// TIA Portal V19 program export: 0 tag tables, 0 data types, 3 data blocks, 24 code blocks (in call order from the OBs), 38 instance data blocks

DATA_BLOCK "time and date"   // DB89
{ S7_Optimized_Access := 'TRUE' }
// stored: MemoryReserve 100
   VAR RETAIN
      "Read time" : DTL;
      "write time" : DTL;
   END_VAR
   VAR
      "Set Time" : Bool;
      day : Int;
      month : Int;
      year : Int;
      hour : Int;
      minute : Int;
   END_VAR
   VAR RETAIN
      "Recipe Start Time" : DTL;
   END_VAR
BEGIN
END_DATA_BLOCK

DATA_BLOCK "IO Mapping"   // DB3
{ S7_Optimized_Access := 'TRUE' }
// stored: MemoryReserve 100
   VAR
      DI : Struct
         "Safety OK" : Bool;
         "IBC Valve is Open" : Bool;
         "IBC Valve is Closed" : Bool;
         "Pump Valve is Open" : Bool;
         "Pump Valve is Closed" : Bool;
         "Flowmeter Feed Valve is Open" : Bool;
         "Flowmerter Feed Valve is Closed" : Bool;
         "Dose Valve is Open" : Bool;
         "Dose Valve is Closed" : Bool;
         "DOL Running Feedback" : Bool;
         "Spare 11" : Bool;
         "Spare 12" : Bool;
         "Spare 13" : Bool;
         "Spare 14" : Bool;
      END_STRUCT;
      DQ : Struct
         "CMD Open IBC Valve" : Bool;
         "CMD Open Pump Feed Valve" : Bool;
         "CMD Open Flowmeter Feed Valve" : Bool;
         "CMD Opend Dosing Valve" : Bool;
         "Run Motor Cooling" : Bool;
         "Spare 6" : Bool;
         "Spare 7" : Bool;
         "Spare 8" : Bool;
         "Spare 9" : Bool;
         "Spare 10" : Bool;
      END_STRUCT;
      AI : Struct
         "Line Pressure" : Int;
         "Buffer level" : Int;
         "Spare 1" : Int;
         "Spare 2" : Int;
      END_STRUCT;
   END_VAR
BEGIN
END_DATA_BLOCK

DATA_BLOCK "HMI Tags"   // DB72
{ S7_Optimized_Access := 'TRUE' }
// stored: MemoryReserve 100
   VAR
      ControlAutoSelect : Bool := FALSE;
      ControlAutoStart : Bool := FALSE;
      ControlAutoStop : Bool := FALSE;
      AutoRunning : Bool := FALSE;
      ResetAlarms : Bool := FALSE;
   END_VAR
   VAR RETAIN
      "Select Input" : Struct
         "Input 1" : Int := 1;
         "Input 2" : Int := 10;
         "Input 3" : Int := 0;
         "Input 4" : Int := 0;
         "Input 5" : Int := 0;
         "Input 6" : Int := 0;
         "Input 7" : Int := 0;
         "Input 8" : Int := 0;
         "Input 9" : Int := 0;
         "Input 10" : Int := 0;
         "Input 11" : Int := 0;
         "Input 12" : Int := 0;
         "Input 13" : Int := 0;
         "Input 14" : Int := 0;
      END_STRUCT;
      "Selected Input" : Struct
         "Input 1" : Int := 0;
         "Input 2" : Int := 0;
         "Input 3" : Int := 0;
         "Input 4" : Int := 0;
         "Input 5" : Int := 0;
         "Input 6" : Int := 0;
         "Input 7" : Int := 0;
         "Input 8" : Int := 0;
         "Input 9" : Int := 0;
         "Input 10" : Int := 0;
         "Input 11" : Int := 0;
         "Input 12" : Int := 0;
         "Input 13" : Int := 0;
         "Input 14" : Int := 0;
      END_STRUCT;
      "Select Output" : Struct
         "output 1" : Int := 0;
         "output 2" : Int := 0;
         "output 3" : Int := 0;
         "output 4" : Int := 0;
         "output 5" : Int := 0;
         "output 6" : Int := 0;
         "output 7" : Int := 0;
         "output 8" : Int := 0;
         "output 9" : Int := 0;
         "output 10" : Int := 0;
      END_STRUCT;
      "Selected Output" : Struct
         "output 1" : Int := 0;
         "output 2" : Int := 0;
         "output 3" : Int := 0;
         "output 4" : Int := 0;
         "output 5" : Int := 0;
         "output 6" : Int := 0;
         "output 7" : Int := 0;
         "output 8" : Int := 0;
         "output 9" : Int := 0;
         "output 10" : Int := 0;
      END_STRUCT;
      LinePressure : "AnalogScale";
      BufferLevel { S7_SetPoint := 'True'} : "AnalogScale";
      SpareAN1 { S7_SetPoint := 'True'} : "AnalogScale";
      SpareAN2 { S7_SetPoint := 'True'} : "AnalogScale";
      CoolOverRunValue { S7_SetPoint := 'True'} : Time := T#1M;
      Pump_Control : "VFD_Control";
   END_VAR
   VAR
      ResetMotorFault : Bool := FALSE;
   END_VAR
   VAR RETAIN
      LinePressureMin { S7_SetPoint := 'True'} : Real := 0.0;
      LinePressureMax : Real := 0.0;
      LinePressureSP : Real := 0.0;
   END_VAR
   VAR
      "Manual Run Motor" : Bool := FALSE;
   END_VAR
   VAR RETAIN
      ModeOneShot : Bool := FALSE;
      ModeRepeat : Bool := TRUE;
      ModeOneShotTime : Bool := FALSE;
      ModeRepeatTime : Bool := FALSE;
      ModeContinous : Bool := FALSE;
   END_VAR
   VAR
      StartDose : Bool := FALSE;
   END_VAR
   VAR RETAIN
      "Required Dose" : Real := 1000.0;
      InflightVal : Real := 0.0;
      CalcDose : Real := 1000.0;
      DoseTime : Time := T#0MS;
      IntervalTime : Time := T#5S;
      IBC : "Valve";
      Flowmeter { S7_SetPoint := 'True'} : "Valve";
      Dose { S7_SetPoint := 'True'} : "Valve";
      Pump { S7_SetPoint := 'True'} : "Valve";
      WriteLogs { S7_SetPoint := 'True'} : Bool := FALSE;
   END_VAR
   VAR
      alarms : DWord := 16#0000_0000;
   END_VAR
   VAR RETAIN
      MinimumLinePressure : Real := 0.0;
      MaximumLinePressure : Real := 12.0;
      SystemEnables : Struct
         "Flowmeter Fitted" : Bool := TRUE;
         LinePressureFitted : Bool := TRUE;
         FlowmeterTemperatureFitted : Bool := TRUE;
         IBCFitted : Bool := FALSE;
         IBCValveFitted : Bool := FALSE;
         FlowmeterValveFitted : Bool := TRUE;
         "Buffer LevelFitted" : Bool := FALSE;
         PumpValveFitted : Bool := FALSE;
         DoseValveFitted : Bool := TRUE;
         ForcedCoolingFitted : Bool := TRUE;
         BufferValveFitted : Bool := FALSE;
      END_STRUCT;
      TemperatureLowSP : Real := 15.0;
      TemperatureHighSP : Real := 30.0;
      BufferHopperMinLVL : Real := 0.0;
      BufferHopperMaxLVL : Real := 0.0;
      BufferHopperLVLSP : Real := 0.0;
      HMISettingsLock : Bool := FALSE;
   END_VAR
   VAR
      DoseState : Int := 0;
   END_VAR
   VAR RETAIN
      DoseWaiting : Time := T#5S;
   END_VAR
   VAR
      FMActualCount : Real := 0.0;
      DoseActTime : Time := T#0MS;
      FmTemperature : Real := 17.8934;
   END_VAR
BEGIN
   LinePressure.AnalogMin := 0;
   LinePressure.AnalogMax := 27648;
   LinePressure.ScaledMIN := 0.0;
   LinePressure.ScaledMax := 11.0;
   LinePressure.ScaledSensor := 0.06127026;
   BufferLevel.AnalogMin := 0;
   BufferLevel.AnalogMax := 0;
   BufferLevel.ScaledMIN := 0.0;
   BufferLevel.ScaledMax := 0.0;
   BufferLevel.ScaledSensor := 0.0;
   SpareAN1.AnalogMin := 0;
   SpareAN1.AnalogMax := 0;
   SpareAN1.ScaledMIN := 0.0;
   SpareAN1.ScaledMax := 0.0;
   SpareAN1.ScaledSensor := 0.0;
   SpareAN2.AnalogMin := 0;
   SpareAN2.AnalogMax := 0;
   SpareAN2.ScaledMIN := 0.0;
   SpareAN2.ScaledMax := 0.0;
   SpareAN2.ScaledSensor := 0.0;
   Pump_Control.NameplateSpeed := 710.0;
   Pump_Control.AutoSpeedSP := 50.0;
   Pump_Control.DriveIsRunning := FALSE;
   Pump_Control.ActualSpeed := 0.0;
   Pump_Control.AxisActive := FALSE;
   Pump_Control.LockoutActive := FALSE;
   Pump_Control.ErrorPResent := FALSE;
   Pump_Control.HMI_VFD_Fault := 0;
   Pump_Control.HMI_Error_Present := FALSE;
   Pump_Control.VFDFaultCode := 0;
   Pump_Control.MotorState := 0;
   Pump_Control.Actual_Current := 0.0007141113;
   Pump_Control.Actual_torque := 0.0;
   Pump_Control.Peak_Current := 0.0;
   Pump_Control.Peak_torque := 0.0;
   IBC.ManOpen := FALSE;
   IBC.FeebackFitted := FALSE;
   IBC.ValveisOpen := FALSE;
   IBC.ValveisClosed := FALSE;
   IBC.ValveAngle := 0.0;
   IBC.FeedbackFaultTime := T#0MS;
   Flowmeter.ManOpen := FALSE;
   Flowmeter.FeebackFitted := FALSE;
   Flowmeter.ValveisOpen := FALSE;
   Flowmeter.ValveisClosed := TRUE;
   Flowmeter.ValveAngle := 90.0;
   Flowmeter.FeedbackFaultTime := T#0MS;
   Dose.ManOpen := FALSE;
   Dose.FeebackFitted := FALSE;
   Dose.ValveisOpen := FALSE;
   Dose.ValveisClosed := TRUE;
   Dose.ValveAngle := 90.0;
   Dose.FeedbackFaultTime := T#0MS;
   Pump.ManOpen := FALSE;
   Pump.FeebackFitted := FALSE;
   Pump.ValveisOpen := FALSE;
   Pump.ValveisClosed := FALSE;
   Pump.ValveAngle := 0.0;
   Pump.FeedbackFaultTime := T#0MS;
END_DATA_BLOCK

ORGANIZATION_BLOCK "Main"   // OB1, LAD, ProgramCycle
TITLE = "Main Program Sweep (Cycle)"
{ S7_Optimized_Access := 'TRUE' }
// stored: SetENOAutomatically false
   VAR_INPUT
      Initial_Call : Bool;   // Initial call of this OB
      Remanence : Bool;   // =True, if remanent data are available
   END_VAR
   VAR_TEMP   // added for the SCL form of the ladder/FBD networks
      _w1 : Bool;
   END_VAR
BEGIN

REGION Network 1: Control
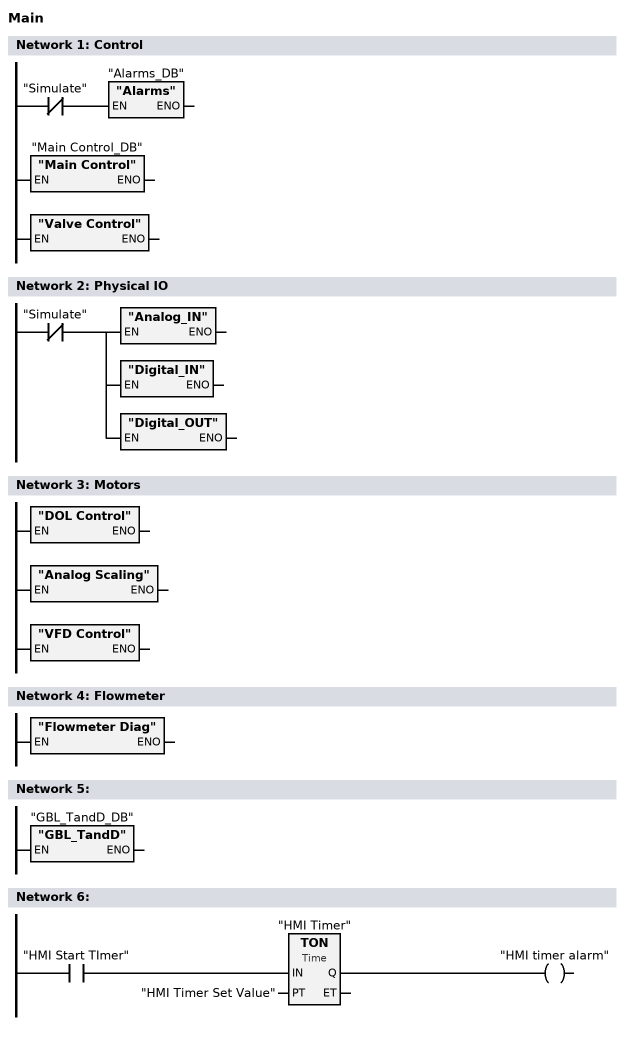
   RUNG wire#powerrail
      I_Contact( "Simulate" )
      "Alarms_DB"()
   END_RUNG
   RUNG wire#powerrail
      "Main Control_DB"()
   END_RUNG
   RUNG wire#powerrail
      "Valve Control"()
   END_RUNG
   // the same network as SCL:
   IF NOT "Simulate" THEN
       "Alarms_DB"();   // "Alarms"
   END_IF;
   "Main Control_DB"();   // "Main Control"
   "Valve Control"();
END_REGION

REGION Network 2: Physical IO
   RUNG wire#powerrail
      I_Contact( "Simulate" )
      wire#w1
      "Analog_IN"()
   END_RUNG
   RUNG wire#w1
      "Digital_IN"()
   END_RUNG
   RUNG wire#w1
      "Digital_OUT"()
   END_RUNG
   // the same network as SCL:
   #_w1 := NOT "Simulate";
   IF #_w1 THEN
       "Analog_IN"();
       "Digital_IN"();
       "Digital_OUT"();
   END_IF;
END_REGION

REGION Network 3: Motors
   RUNG wire#powerrail
      "DOL Control"()
   END_RUNG
   RUNG wire#powerrail
      "Analog Scaling"()
   END_RUNG
   RUNG wire#powerrail
      "VFD Control"()
   END_RUNG
   // the same network as SCL:
   "DOL Control"();
   "Analog Scaling"();
   "VFD Control"();
END_REGION

REGION Network 4: Flowmeter
   RUNG wire#powerrail
      "Flowmeter Diag"()
   END_RUNG
   // the same network as SCL:
   "Flowmeter Diag"();
END_REGION

REGION Network 5
   RUNG wire#powerrail
      "GBL_TandD_DB"()
   END_RUNG
   // the same network as SCL:
   "GBL_TandD_DB"();   // "GBL_TandD"
END_REGION

REGION Network 6
   RUNG wire#powerrail
      Contact( "HMI Start TImer" )
      { S7_Templates := "time_type := Time" } "HMI Timer".TON(pt := "HMI Timer Set Value", et =>)
      Coil( "HMI timer alarm" )
   END_RUNG
   // the same network as SCL:
   "HMI Timer".TON(IN := "HMI Start TImer", PT := "HMI Timer Set Value");
   "HMI timer alarm" := "HMI Timer".Q;
END_REGION
END_ORGANIZATION_BLOCK

FUNCTION_BLOCK "Alarms"   // FB7, LAD
{ S7_Optimized_Access := 'TRUE' }
// stored: MemoryReserve 100, SetENOAutomatically false
   VAR_TEMP   // added for the SCL form of the ladder/FBD networks
      _w1 : Bool;
      _w2 : Bool;
      _w3 : Bool;
   END_VAR
BEGIN

REGION Network 1: IBC Valve Open Fault
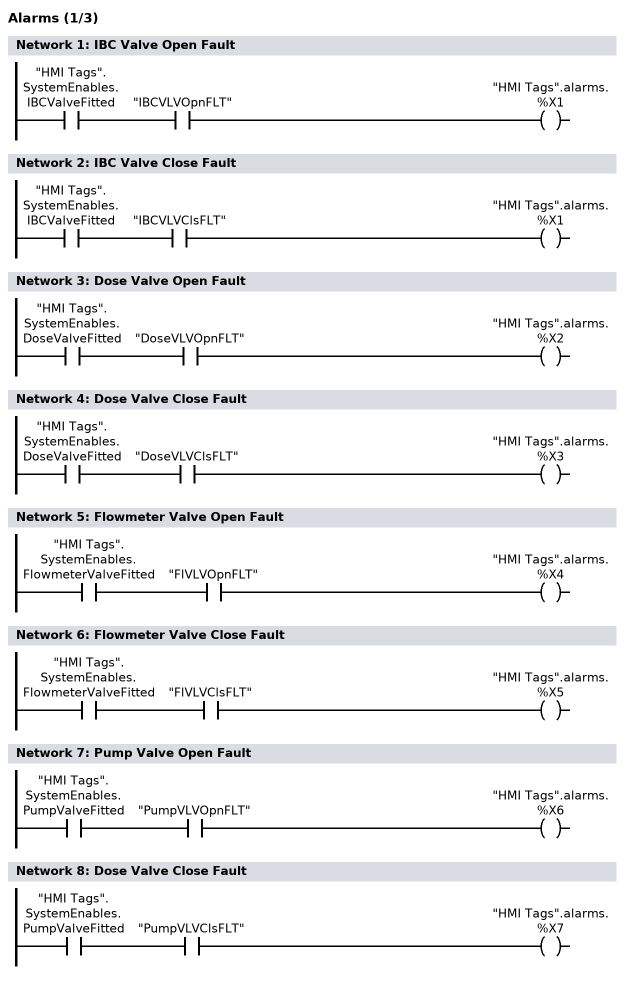
   RUNG wire#powerrail
      Contact( "HMI Tags".SystemEnables.IBCValveFitted )
      Contact( "IBCVLVOpnFLT" )
      Coil( "HMI Tags".alarms.%X1 )
   END_RUNG
   // the same network as SCL:
   "HMI Tags".alarms.%X1 := "HMI Tags".SystemEnables.IBCValveFitted AND "IBCVLVOpnFLT";
END_REGION

REGION Network 2: IBC Valve Close Fault
   RUNG wire#powerrail
      Contact( "HMI Tags".SystemEnables.IBCValveFitted )
      Contact( "IBCVLVClsFLT" )
      Coil( "HMI Tags".alarms.%X1 )
   END_RUNG
   // the same network as SCL:
   "HMI Tags".alarms.%X1 := "HMI Tags".SystemEnables.IBCValveFitted AND "IBCVLVClsFLT";
END_REGION

REGION Network 3: Dose Valve Open Fault
   RUNG wire#powerrail
      Contact( "HMI Tags".SystemEnables.DoseValveFitted )
      Contact( "DoseVLVOpnFLT" )
      Coil( "HMI Tags".alarms.%X2 )
   END_RUNG
   // the same network as SCL:
   "HMI Tags".alarms.%X2 := "HMI Tags".SystemEnables.DoseValveFitted AND "DoseVLVOpnFLT";
END_REGION

REGION Network 4: Dose Valve Close Fault
   RUNG wire#powerrail
      Contact( "HMI Tags".SystemEnables.DoseValveFitted )
      Contact( "DoseVLVClsFLT" )
      Coil( "HMI Tags".alarms.%X3 )
   END_RUNG
   // the same network as SCL:
   "HMI Tags".alarms.%X3 := "HMI Tags".SystemEnables.DoseValveFitted AND "DoseVLVClsFLT";
END_REGION

REGION Network 5: Flowmeter Valve Open Fault
   RUNG wire#powerrail
      Contact( "HMI Tags".SystemEnables.FlowmeterValveFitted )
      Contact( "FlVLVOpnFLT" )
      Coil( "HMI Tags".alarms.%X4 )
   END_RUNG
   // the same network as SCL:
   "HMI Tags".alarms.%X4 := "HMI Tags".SystemEnables.FlowmeterValveFitted AND "FlVLVOpnFLT";
END_REGION

REGION Network 6: Flowmeter Valve Close Fault
   RUNG wire#powerrail
      Contact( "HMI Tags".SystemEnables.FlowmeterValveFitted )
      Contact( "FlVLVClsFLT" )
      Coil( "HMI Tags".alarms.%X5 )
   END_RUNG
   // the same network as SCL:
   "HMI Tags".alarms.%X5 := "HMI Tags".SystemEnables.FlowmeterValveFitted AND "FlVLVClsFLT";
END_REGION

REGION Network 7: Pump Valve Open Fault
   RUNG wire#powerrail
      Contact( "HMI Tags".SystemEnables.PumpValveFitted )
      Contact( "PumpVLVOpnFLT" )
      Coil( "HMI Tags".alarms.%X6 )
   END_RUNG
   // the same network as SCL:
   "HMI Tags".alarms.%X6 := "HMI Tags".SystemEnables.PumpValveFitted AND "PumpVLVOpnFLT";
END_REGION

REGION Network 8: Dose Valve Close Fault
   RUNG wire#powerrail
      Contact( "HMI Tags".SystemEnables.PumpValveFitted )
      Contact( "PumpVLVClsFLT" )
      Coil( "HMI Tags".alarms.%X7 )
   END_RUNG
   // the same network as SCL:
   "HMI Tags".alarms.%X7 := "HMI Tags".SystemEnables.PumpValveFitted AND "PumpVLVClsFLT";
END_REGION

REGION Network 9: Flowmeter not counting when required
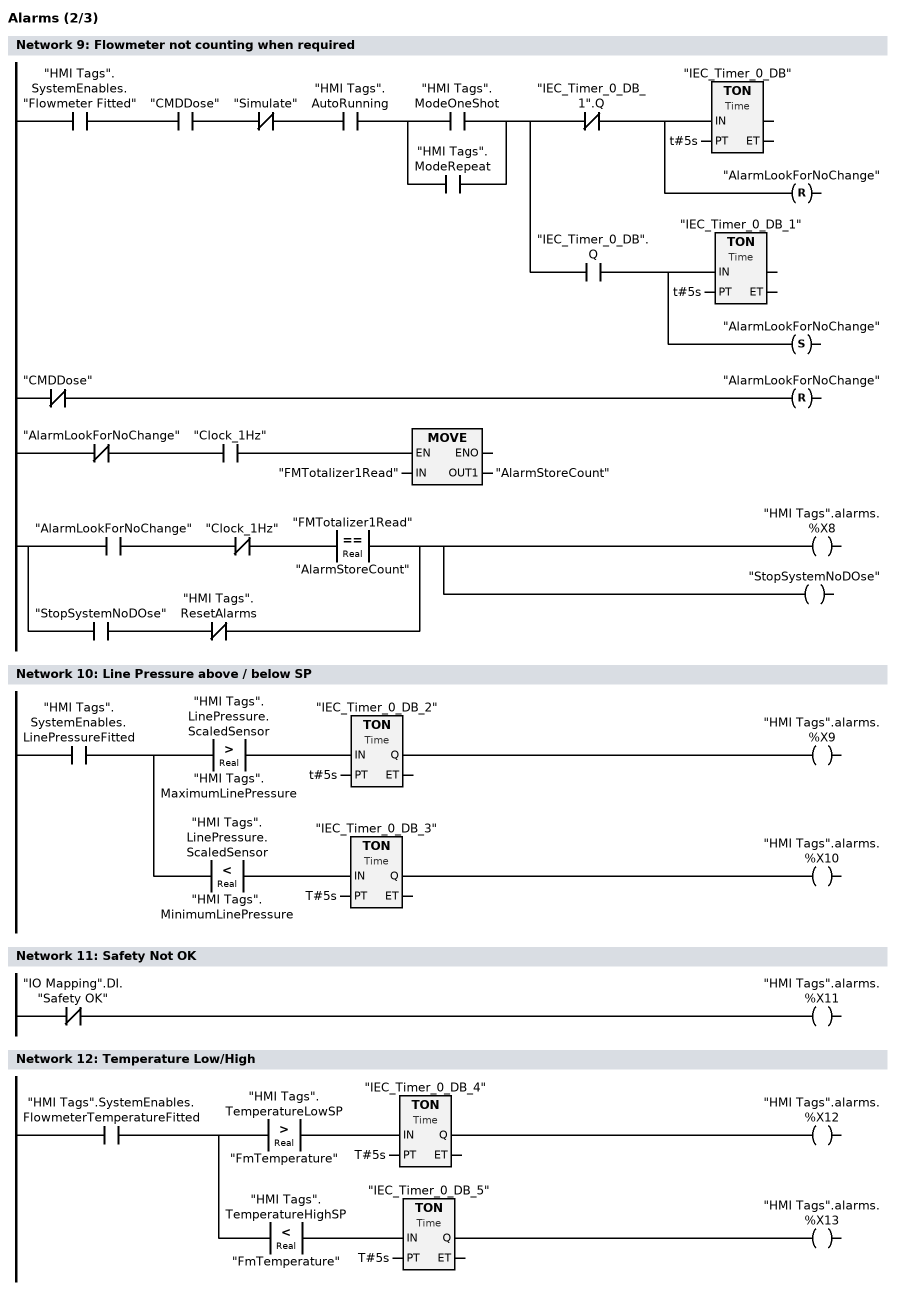
   RUNG wire#powerrail
      Contact( "HMI Tags".SystemEnables."Flowmeter Fitted" )
      Contact( "CMDDose" )
      I_Contact( "Simulate" )
      Contact( "HMI Tags".AutoRunning )
      wire#w1
      Contact( "HMI Tags".ModeOneShot )
      wire#w2
      I_Contact( "IEC_Timer_0_DB_1".Q )
      wire#w3
      { S7_Templates := "time_type := Time" } "IEC_Timer_0_DB".TON(pt := t#5s, et =>)
   END_RUNG
   RUNG wire#w1
      Contact( "HMI Tags".ModeRepeat )
   END_RUNG wire#w2
   RUNG wire#w3
      R_Coil( "AlarmLookForNoChange" )
   END_RUNG
   RUNG wire#w2
      Contact( "IEC_Timer_0_DB".Q )
      wire#w4
      { S7_Templates := "time_type := Time" } "IEC_Timer_0_DB_1".TON(pt := t#5s, et =>)
   END_RUNG
   RUNG wire#w4
      S_Coil( "AlarmLookForNoChange" )
   END_RUNG
   RUNG wire#powerrail
      I_Contact( "CMDDose" )
      R_Coil( "AlarmLookForNoChange" )
   END_RUNG
   RUNG wire#powerrail
      I_Contact( "AlarmLookForNoChange" )
      Contact( "Clock_1Hz" )
      Move(in := "FMTotalizer1Read", out1 => "AlarmStoreCount")
   END_RUNG
   RUNG wire#powerrail
      Contact( "AlarmLookForNoChange" )
      I_Contact( "Clock_1Hz" )
      { S7_Templates := "SrcType := Real" } EQ_Contact(in1 := "FMTotalizer1Read", in2 := "AlarmStoreCount")
      wire#w5
      Coil( "HMI Tags".alarms.%X8 )
   END_RUNG
   RUNG wire#powerrail
      Contact( "StopSystemNoDOse" )
      I_Contact( "HMI Tags".ResetAlarms )
   END_RUNG wire#w5
   RUNG wire#w5
      Coil( "StopSystemNoDOse" )
   END_RUNG
   // the same network as SCL:
   #_w1 := "HMI Tags".SystemEnables."Flowmeter Fitted" AND "CMDDose" AND NOT "Simulate" AND "HMI Tags".AutoRunning AND ("HMI Tags".ModeOneShot OR "HMI Tags".ModeRepeat);
   #_w2 := #_w1 AND NOT "IEC_Timer_0_DB_1".Q;
   "IEC_Timer_0_DB".TON(IN := #_w2, PT := t#5s);
   IF #_w2 THEN "AlarmLookForNoChange" := FALSE; END_IF;
   #_w3 := #_w1 AND "IEC_Timer_0_DB".Q;
   "IEC_Timer_0_DB_1".TON(IN := #_w3, PT := t#5s);
   IF #_w3 THEN "AlarmLookForNoChange" := TRUE; END_IF;
   IF NOT "CMDDose" THEN "AlarmLookForNoChange" := FALSE; END_IF;
   IF NOT "AlarmLookForNoChange" AND "Clock_1Hz" THEN "AlarmStoreCount" := "FMTotalizer1Read"; END_IF;
   "HMI Tags".alarms.%X8 := ("AlarmLookForNoChange" AND NOT "Clock_1Hz" AND ("FMTotalizer1Read" = "AlarmStoreCount")) OR ("StopSystemNoDOse" AND NOT "HMI Tags".ResetAlarms);
   "StopSystemNoDOse" := "HMI Tags".alarms.%X8;
END_REGION

REGION Network 10: Line Pressure above / below SP
   RUNG wire#powerrail
      Contact( "HMI Tags".SystemEnables.LinePressureFitted )
      wire#w1
      { S7_Templates := "SrcType := Real" } GT_Contact(in1 := "HMI Tags".LinePressure.ScaledSensor, in2 := "HMI Tags".MaximumLinePressure)
      { S7_Templates := "time_type := Time" } "IEC_Timer_0_DB_2".TON(pt := t#5s, et =>)
      Coil( "HMI Tags".alarms.%X9 )
   END_RUNG
   RUNG wire#w1
      { S7_Templates := "SrcType := Real" } LT_Contact(in1 := "HMI Tags".LinePressure.ScaledSensor, in2 := "HMI Tags".MinimumLinePressure)
      { S7_Templates := "time_type := Time" } "IEC_Timer_0_DB_3".TON(pt := T#5s, et =>)
      Coil( "HMI Tags".alarms.%X10 )
   END_RUNG
   // the same network as SCL:
   "IEC_Timer_0_DB_2".TON(IN := "HMI Tags".SystemEnables.LinePressureFitted AND ("HMI Tags".LinePressure.ScaledSensor > "HMI Tags".MaximumLinePressure),
                          PT := t#5s);
   "HMI Tags".alarms.%X9 := "IEC_Timer_0_DB_2".Q;
   "IEC_Timer_0_DB_3".TON(IN := "HMI Tags".SystemEnables.LinePressureFitted AND ("HMI Tags".LinePressure.ScaledSensor < "HMI Tags".MinimumLinePressure),
                          PT := T#5s);
   "HMI Tags".alarms.%X10 := "IEC_Timer_0_DB_3".Q;
END_REGION

REGION Network 11: Safety Not OK
   RUNG wire#powerrail
      I_Contact( "IO Mapping".DI."Safety OK" )
      Coil( "HMI Tags".alarms.%X11 )
   END_RUNG
   // the same network as SCL:
   "HMI Tags".alarms.%X11 := NOT "IO Mapping".DI."Safety OK";
END_REGION

REGION Network 12: Temperature Low/High
   RUNG wire#powerrail
      Contact( "HMI Tags".SystemEnables.FlowmeterTemperatureFitted )
      wire#w1
      { S7_Templates := "SrcType := Real" } GT_Contact(in1 := "HMI Tags".TemperatureLowSP, in2 := "FmTemperature")
      { S7_Templates := "time_type := Time" } "IEC_Timer_0_DB_4".TON(pt := T#5s, et =>)
      Coil( "HMI Tags".alarms.%X12 )
   END_RUNG
   RUNG wire#w1
      { S7_Templates := "SrcType := Real" } LT_Contact(in1 := "HMI Tags".TemperatureHighSP, in2 := "FmTemperature")
      { S7_Templates := "time_type := Time" } "IEC_Timer_0_DB_5".TON(pt := T#5s, et =>)
      Coil( "HMI Tags".alarms.%X13 )
   END_RUNG
   // the same network as SCL:
   "IEC_Timer_0_DB_4".TON(IN := "HMI Tags".SystemEnables.FlowmeterTemperatureFitted AND ("HMI Tags".TemperatureLowSP > "FmTemperature"),
                          PT := T#5s);
   "HMI Tags".alarms.%X12 := "IEC_Timer_0_DB_4".Q;
   "IEC_Timer_0_DB_5".TON(IN := "HMI Tags".SystemEnables.FlowmeterTemperatureFitted AND ("HMI Tags".TemperatureHighSP < "FmTemperature"),
                          PT := T#5s);
   "HMI Tags".alarms.%X13 := "IEC_Timer_0_DB_5".Q;
END_REGION

REGION Network 13: VFDFAULT
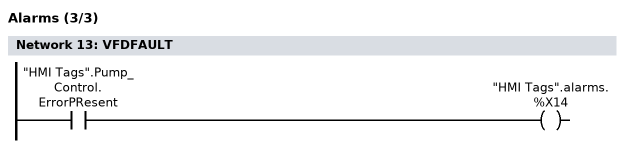
   RUNG wire#powerrail
      Contact( "HMI Tags".Pump_Control.ErrorPResent )
      Coil( "HMI Tags".alarms.%X14 )
   END_RUNG
   // the same network as SCL:
   "HMI Tags".alarms.%X14 := "HMI Tags".Pump_Control.ErrorPResent;
END_REGION
END_FUNCTION_BLOCK

FUNCTION_BLOCK "Main Control"   // FB1, LAD
{ S7_Optimized_Access := 'TRUE' }
// stored: MemoryReserve 100, SetENOAutomatically false
   VAR
      store : Bool;
   END_VAR
   VAR_TEMP   // added for the SCL form of the ladder/FBD networks
      _w1 : Bool;
      _w2 : Bool;
   END_VAR
BEGIN

REGION Network 1: Control Auto Run
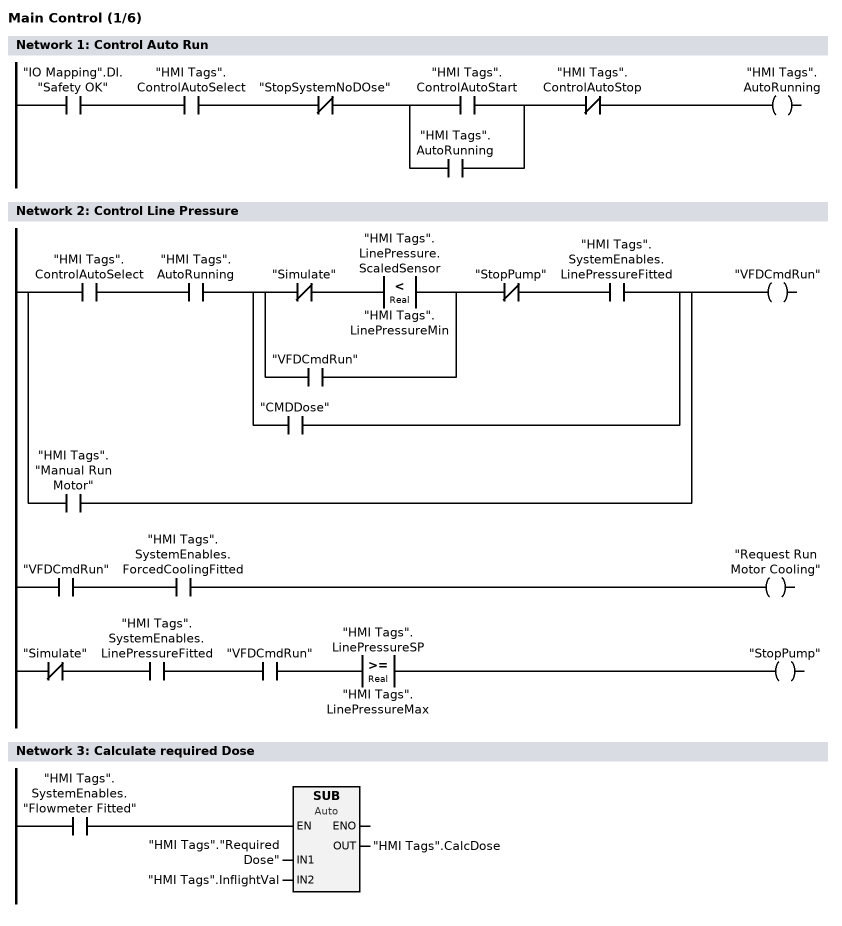
   RUNG wire#powerrail
      Contact( "IO Mapping".DI."Safety OK" )
      Contact( "HMI Tags".ControlAutoSelect )
      I_Contact( "StopSystemNoDOse" )
      wire#w1
      Contact( "HMI Tags".ControlAutoStart )
      wire#w2
      I_Contact( "HMI Tags".ControlAutoStop )
      Coil( "HMI Tags".AutoRunning )
   END_RUNG
   RUNG wire#w1
      Contact( "HMI Tags".AutoRunning )
   END_RUNG wire#w2
   // the same network as SCL:
   "HMI Tags".AutoRunning := "IO Mapping".DI."Safety OK" AND "HMI Tags".ControlAutoSelect AND NOT "StopSystemNoDOse" AND ("HMI Tags".ControlAutoStart OR "HMI Tags".AutoRunning) AND NOT "HMI Tags".ControlAutoStop;
END_REGION

REGION Network 2: Control Line Pressure
   RUNG wire#powerrail
      Contact( "HMI Tags".ControlAutoSelect )
      Contact( "HMI Tags".AutoRunning )
      wire#w1
      I_Contact( "Simulate" )
      { S7_Templates := "SrcType := Real" } LT_Contact(in1 := "HMI Tags".LinePressure.ScaledSensor, in2 := "HMI Tags".LinePressureMin)
      wire#w2
      I_Contact( "StopPump" )
      Contact( "HMI Tags".SystemEnables.LinePressureFitted )
      wire#w3
      Coil( "VFDCmdRun" )
   END_RUNG
   RUNG wire#w1
      Contact( "VFDCmdRun" )
   END_RUNG wire#w2
   RUNG wire#w1
      Contact( "CMDDose" )
   END_RUNG wire#w3
   RUNG wire#powerrail
      Contact( "HMI Tags"."Manual Run Motor" )
   END_RUNG wire#w3
   RUNG wire#powerrail
      Contact( "VFDCmdRun" )
      Contact( "HMI Tags".SystemEnables.ForcedCoolingFitted )
      Coil( "Request Run Motor Cooling" )
   END_RUNG
   RUNG wire#powerrail
      I_Contact( "Simulate" )
      Contact( "HMI Tags".SystemEnables.LinePressureFitted )
      Contact( "VFDCmdRun" )
      { S7_Templates := "SrcType := Real" } GE_Contact(in1 := "HMI Tags".LinePressureSP, in2 := "HMI Tags".LinePressureMax)
      Coil( "StopPump" )
   END_RUNG
   // the same network as SCL:
   "VFDCmdRun" := ("HMI Tags".ControlAutoSelect AND "HMI Tags".AutoRunning AND ((((NOT "Simulate" AND ("HMI Tags".LinePressure.ScaledSensor < "HMI Tags".LinePressureMin)) OR "VFDCmdRun") AND NOT "StopPump" AND "HMI Tags".SystemEnables.LinePressureFitted) OR "CMDDose")) OR "HMI Tags"."Manual Run Motor";
   "Request Run Motor Cooling" := "VFDCmdRun" AND "HMI Tags".SystemEnables.ForcedCoolingFitted;
   "StopPump" := NOT "Simulate" AND "HMI Tags".SystemEnables.LinePressureFitted AND "VFDCmdRun" AND ("HMI Tags".LinePressureSP >= "HMI Tags".LinePressureMax);
END_REGION

REGION Network 3: Calculate required Dose
   RUNG wire#powerrail
      Contact( "HMI Tags".SystemEnables."Flowmeter Fitted" )
      Sub(in1 := "HMI Tags"."Required Dose", in2 := "HMI Tags".InflightVal, out => "HMI Tags".CalcDose)
   END_RUNG
   // the same network as SCL:
   IF "HMI Tags".SystemEnables."Flowmeter Fitted" THEN
       "HMI Tags".CalcDose := "HMI Tags"."Required Dose" - "HMI Tags".InflightVal;
   END_IF;
END_REGION

REGION Network 4: Open Valves to Dose
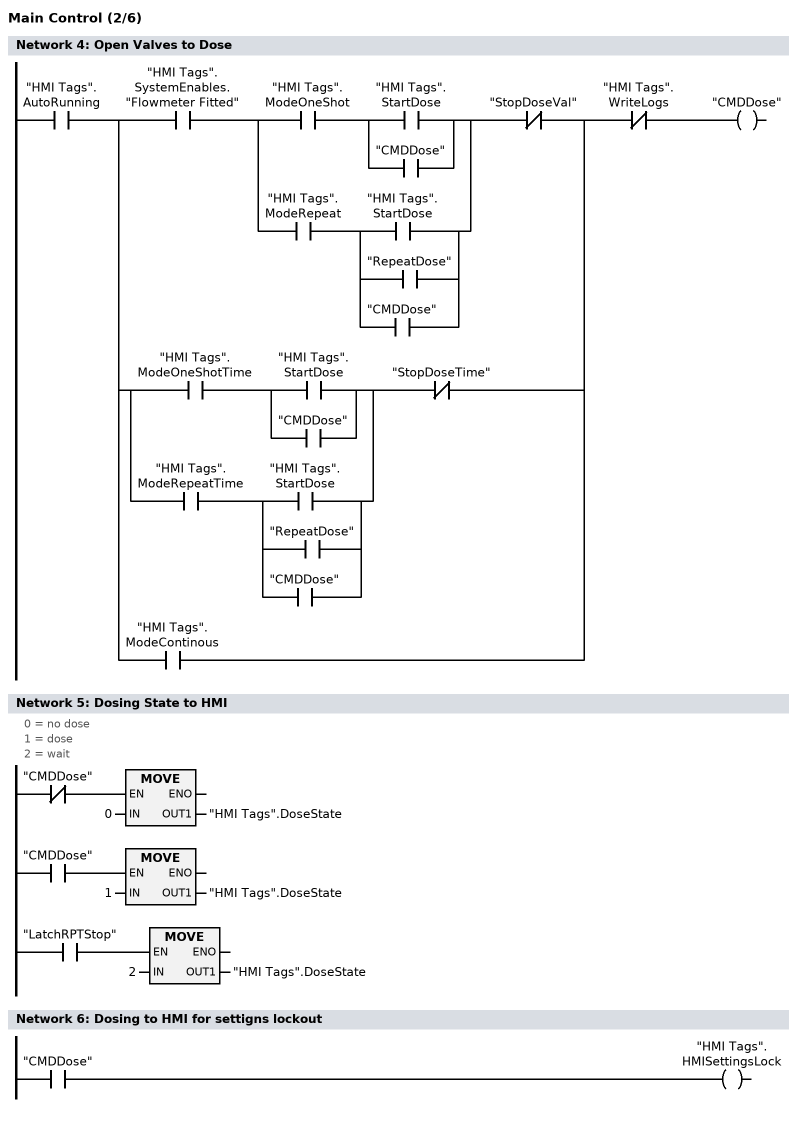
   RUNG wire#powerrail
      Contact( "HMI Tags".AutoRunning )
      wire#w1
      Contact( "HMI Tags".SystemEnables."Flowmeter Fitted" )
      wire#w2
      Contact( "HMI Tags".ModeOneShot )
      wire#w3
      Contact( "HMI Tags".StartDose )
      wire#w4
      I_Contact( "StopDoseVal" )
      wire#w6
      I_Contact( "HMI Tags".WriteLogs )
      Coil( "CMDDose" )
   END_RUNG
   RUNG wire#w3
      Contact( "CMDDose" )
   END_RUNG wire#w4
   RUNG wire#w2
      Contact( "HMI Tags".ModeRepeat )
      wire#w5
      Contact( "HMI Tags".StartDose )
   END_RUNG wire#w4
   RUNG wire#w5
      Contact( "RepeatDose" )
   END_RUNG wire#w4
   RUNG wire#w5
      Contact( "CMDDose" )
   END_RUNG wire#w4
   RUNG wire#w1
      Contact( "HMI Tags".ModeOneShotTime )
      wire#w7
      Contact( "HMI Tags".StartDose )
      wire#w8
      I_Contact( "StopDoseTime" )
   END_RUNG wire#w6
   RUNG wire#w7
      Contact( "CMDDose" )
   END_RUNG wire#w8
   RUNG wire#w1
      Contact( "HMI Tags".ModeRepeatTime )
      wire#w9
      Contact( "HMI Tags".StartDose )
   END_RUNG wire#w8
   RUNG wire#w9
      Contact( "RepeatDose" )
   END_RUNG wire#w8
   RUNG wire#w9
      Contact( "CMDDose" )
   END_RUNG wire#w8
   RUNG wire#w1
      Contact( "HMI Tags".ModeContinous )
   END_RUNG wire#w6
   // the same network as SCL:
   "CMDDose" := "HMI Tags".AutoRunning AND (("HMI Tags".SystemEnables."Flowmeter Fitted" AND (("HMI Tags".ModeOneShot AND ("HMI Tags".StartDose OR "CMDDose")) OR ("HMI Tags".ModeRepeat AND ("HMI Tags".StartDose OR "RepeatDose" OR "CMDDose"))) AND NOT "StopDoseVal") OR ((("HMI Tags".ModeOneShotTime AND ("HMI Tags".StartDose OR "CMDDose")) OR ("HMI Tags".ModeRepeatTime AND ("HMI Tags".StartDose OR "RepeatDose" OR "CMDDose"))) AND NOT "StopDoseTime") OR "HMI Tags".ModeContinous) AND NOT "HMI Tags".WriteLogs;
END_REGION

REGION Network 5: Dosing State to HMI
   // 0 = no dose
   // 1 = dose
   // 2 = wait
   RUNG wire#powerrail
      I_Contact( "CMDDose" )
      Move(in := 0, out1 => "HMI Tags".DoseState)
   END_RUNG
   RUNG wire#powerrail
      Contact( "CMDDose" )
      Move(in := 1, out1 => "HMI Tags".DoseState)
   END_RUNG
   RUNG wire#powerrail
      Contact( "LatchRPTStop" )
      Move(in := 2, out1 => "HMI Tags".DoseState)
   END_RUNG
   // the same network as SCL:
   IF NOT "CMDDose" THEN "HMI Tags".DoseState := 0; END_IF;
   IF "CMDDose" THEN "HMI Tags".DoseState := 1; END_IF;
   IF "LatchRPTStop" THEN "HMI Tags".DoseState := 2; END_IF;
END_REGION

REGION Network 6: Dosing to HMI for settigns lockout
   RUNG wire#powerrail
      Contact( "CMDDose" )
      Coil( "HMI Tags".HMISettingsLock )
   END_RUNG
   // the same network as SCL:
   "HMI Tags".HMISettingsLock := "CMDDose";
END_REGION

REGION Network 7: Command the flowmeter to count
   // This should start the flowmeter counting slightly ahead of opening the valves.
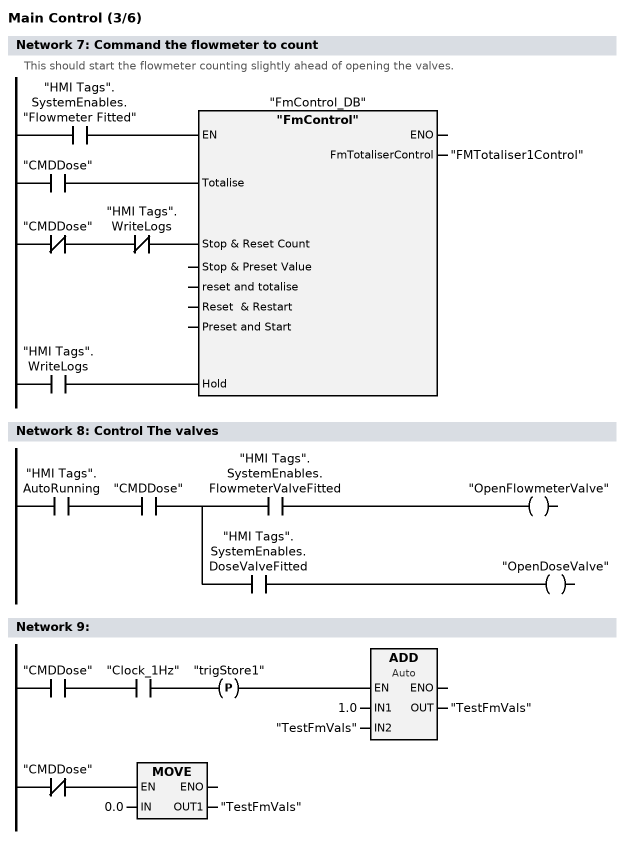
   RUNG wire#powerrail
      Contact( "HMI Tags".SystemEnables."Flowmeter Fitted" )
      "FmControl_DB"(Totalise := wire#w1, "Stop & Reset Count" := wire#w2, Hold := wire#w3, "Stop & Preset Value" :=, "reset and totalise" :=, "Reset  & Restart" :=, "Preset and Start" :=, FmTotaliserControl => "FMTotaliser1Control")
   END_RUNG
   RUNG wire#powerrail
      Contact( "CMDDose" )
   END_RUNG wire#w1
   RUNG wire#powerrail
      I_Contact( "CMDDose" )
      I_Contact( "HMI Tags".WriteLogs )
   END_RUNG wire#w2
   RUNG wire#powerrail
      Contact( "HMI Tags".WriteLogs )
   END_RUNG wire#w3
   // the same network as SCL:
   IF "HMI Tags".SystemEnables."Flowmeter Fitted" THEN
       "FmControl_DB"(Totalise := "CMDDose",   // "FmControl"
                      "Stop & Reset Count" := NOT "CMDDose" AND NOT "HMI Tags".WriteLogs,
                      Hold := "HMI Tags".WriteLogs,
                      FmTotaliserControl => "FMTotaliser1Control");
   END_IF;
END_REGION

REGION Network 8: Control The valves
   RUNG wire#powerrail
      Contact( "HMI Tags".AutoRunning )
      Contact( "CMDDose" )
      wire#w1
      Contact( "HMI Tags".SystemEnables.FlowmeterValveFitted )
      Coil( "OpenFlowmeterValve" )
   END_RUNG
   RUNG wire#w1
      Contact( "HMI Tags".SystemEnables.DoseValveFitted )
      Coil( "OpenDoseValve" )
   END_RUNG
   // the same network as SCL:
   #_w1 := "HMI Tags".AutoRunning AND "CMDDose";
   "OpenFlowmeterValve" := #_w1 AND "HMI Tags".SystemEnables.FlowmeterValveFitted;
   "OpenDoseValve" := #_w1 AND "HMI Tags".SystemEnables.DoseValveFitted;
END_REGION

REGION Network 9
   RUNG wire#powerrail
      Contact( "CMDDose" )
      Contact( "Clock_1Hz" )
      P_Trig( "trigStore1" )
      Add(in1 := 1.0, in2 := "TestFmVals", out => "TestFmVals")
   END_RUNG
   RUNG wire#powerrail
      I_Contact( "CMDDose" )
      Move(in := 0.0, out1 => "TestFmVals")
   END_RUNG
   // the same network as SCL:
   #_w1 := "CMDDose" AND "Clock_1Hz";
   #_w2 := #_w1 AND NOT "trigStore1";   // rising edge
   "trigStore1" := #_w1;
   IF #_w2 THEN "TestFmVals" := 1.0 + "TestFmVals"; END_IF;
   IF NOT "CMDDose" THEN "TestFmVals" := 0.0; END_IF;
END_REGION

REGION Network 10: Wait for flow Value OneShot value or time
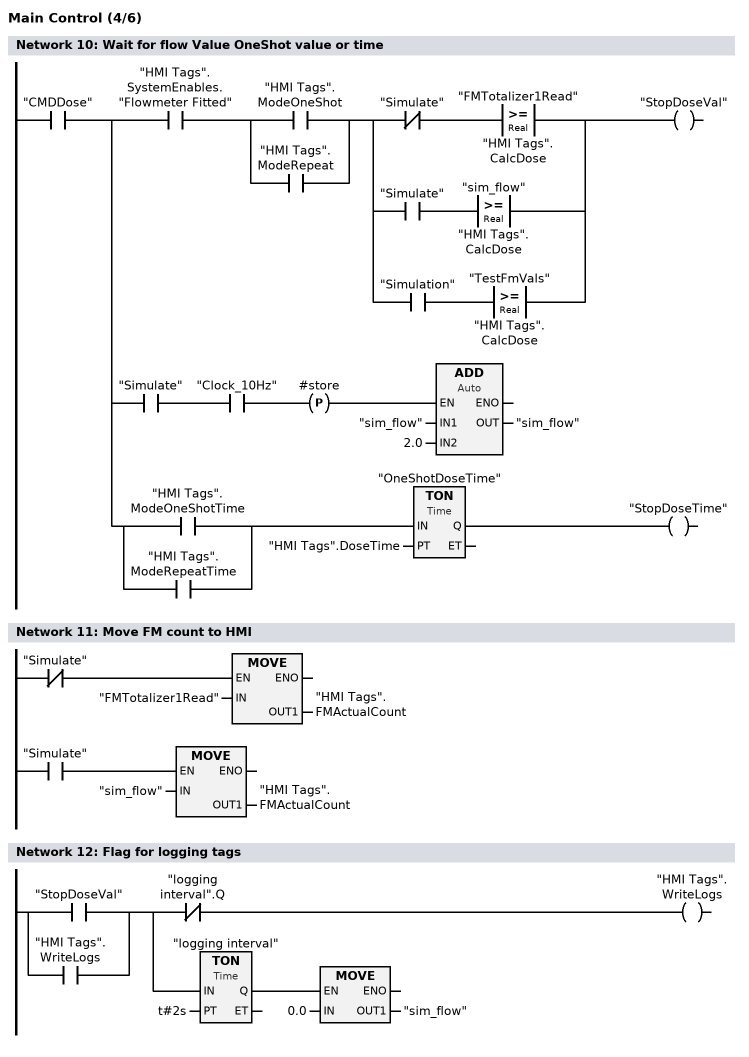
   RUNG wire#powerrail
      Contact( "CMDDose" )
      wire#w1
      Contact( "HMI Tags".SystemEnables."Flowmeter Fitted" )
      wire#w2
      Contact( "HMI Tags".ModeOneShot )
      wire#w3
      I_Contact( "Simulate" )
      { S7_Templates := "SrcType := Real" } GE_Contact(in1 := "FMTotalizer1Read", in2 := "HMI Tags".CalcDose)
      wire#w4
      Coil( "StopDoseVal" )
   END_RUNG
   RUNG wire#w2
      Contact( "HMI Tags".ModeRepeat )
   END_RUNG wire#w3
   RUNG wire#w3
      Contact( "Simulate" )
      { S7_Templates := "SrcType := Real" } GE_Contact(in1 := "sim_flow", in2 := "HMI Tags".CalcDose)
   END_RUNG wire#w4
   RUNG wire#w3
      Contact( "Simulation" )
      { S7_Templates := "SrcType := Real" } GE_Contact(in1 := "TestFmVals", in2 := "HMI Tags".CalcDose)
   END_RUNG wire#w4
   RUNG wire#w1
      Contact( "Simulate" )
      Contact( "Clock_10Hz" )
      P_Trig( #store )
      Add(in1 := "sim_flow", in2 := 2.0, out => "sim_flow")
   END_RUNG
   RUNG wire#w1
      Contact( "HMI Tags".ModeOneShotTime )
      wire#w5
      { S7_Templates := "time_type := Time" } "OneShotDoseTime".TON(pt := "HMI Tags".DoseTime, et =>)
      Coil( "StopDoseTime" )
   END_RUNG
   RUNG wire#w1
      Contact( "HMI Tags".ModeRepeatTime )
   END_RUNG wire#w5
   // the same network as SCL:
   "StopDoseVal" := "CMDDose" AND "HMI Tags".SystemEnables."Flowmeter Fitted" AND ("HMI Tags".ModeOneShot OR "HMI Tags".ModeRepeat) AND ((NOT "Simulate" AND ("FMTotalizer1Read" >= "HMI Tags".CalcDose)) OR ("Simulate" AND ("sim_flow" >= "HMI Tags".CalcDose)) OR ("Simulation" AND ("TestFmVals" >= "HMI Tags".CalcDose)));
   #_w1 := "CMDDose" AND "Simulate" AND "Clock_10Hz";
   #_w2 := #_w1 AND NOT #store;   // rising edge
   #store := #_w1;
   IF #_w2 THEN "sim_flow" := "sim_flow" + 2.0; END_IF;
   "OneShotDoseTime".TON(IN := "CMDDose" AND ("HMI Tags".ModeOneShotTime OR "HMI Tags".ModeRepeatTime),
                         PT := "HMI Tags".DoseTime);
   "StopDoseTime" := "OneShotDoseTime".Q;
END_REGION

REGION Network 11: Move FM count to HMI
   RUNG wire#powerrail
      I_Contact( "Simulate" )
      Move(in := "FMTotalizer1Read", out1 => "HMI Tags".FMActualCount)
   END_RUNG
   RUNG wire#powerrail
      Contact( "Simulate" )
      Move(in := "sim_flow", out1 => "HMI Tags".FMActualCount)
   END_RUNG
   // the same network as SCL:
   IF NOT "Simulate" THEN "HMI Tags".FMActualCount := "FMTotalizer1Read"; END_IF;
   IF "Simulate" THEN "HMI Tags".FMActualCount := "sim_flow"; END_IF;
END_REGION

REGION Network 12: Flag for logging tags
   RUNG wire#powerrail
      Contact( "StopDoseVal" )
      wire#w1
      I_Contact( "logging interval".Q )
      Coil( "HMI Tags".WriteLogs )
   END_RUNG
   RUNG wire#powerrail
      Contact( "HMI Tags".WriteLogs )
   END_RUNG wire#w1
   RUNG wire#w1
      { S7_Templates := "time_type := Time" } "logging interval".TON(pt := t#2s, et =>)
      Move(in := 0.0, out1 => "sim_flow")
   END_RUNG
   // the same network as SCL:
   #_w1 := "StopDoseVal" OR "HMI Tags".WriteLogs;
   "HMI Tags".WriteLogs := #_w1 AND NOT "logging interval".Q;
   "logging interval".TON(IN := #_w1, PT := t#2s);
   IF "logging interval".Q THEN "sim_flow" := 0.0; END_IF;
END_REGION

REGION Network 13: Repeat Dose After Time
   // Latch dose start and dose stop for repeat doses then unlatch on the next dose
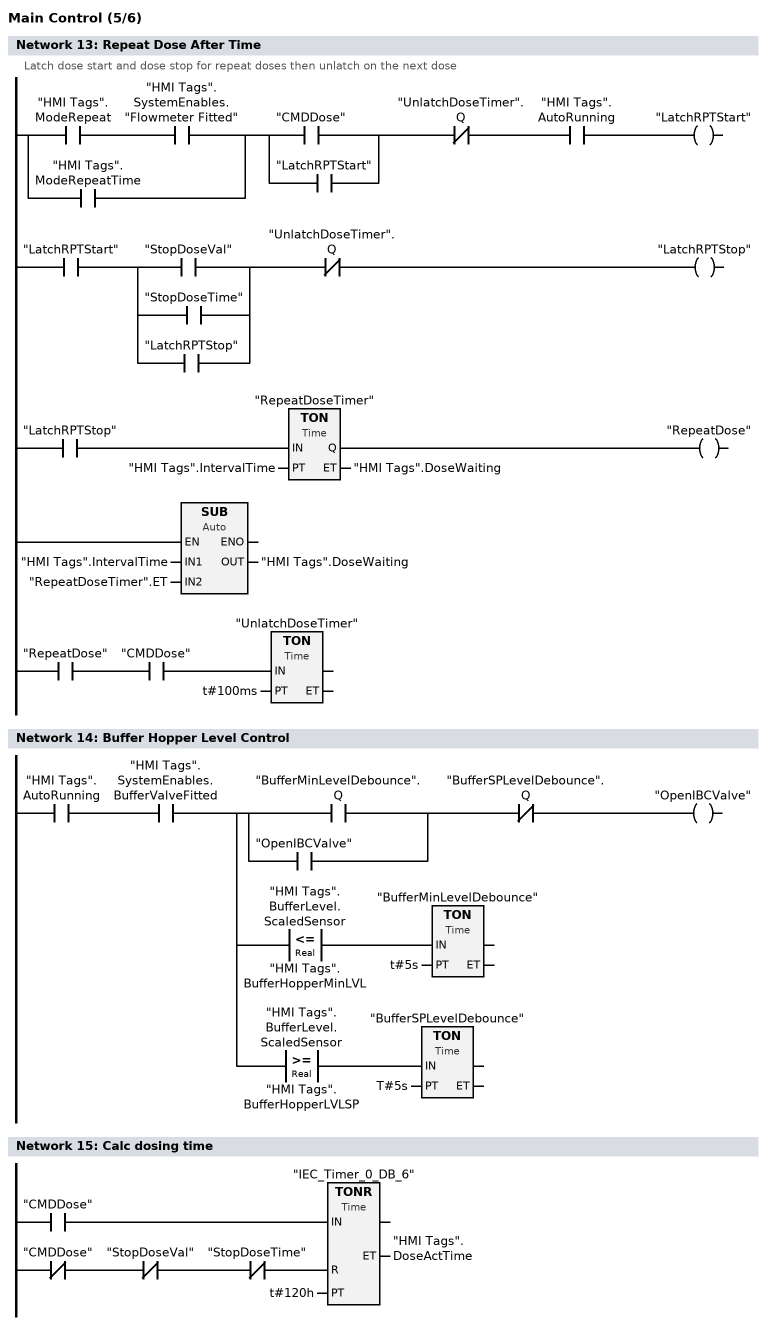
   RUNG wire#powerrail
      Contact( "HMI Tags".ModeRepeat )
      Contact( "HMI Tags".SystemEnables."Flowmeter Fitted" )
      wire#w1
      Contact( "CMDDose" )
      wire#w2
      I_Contact( "UnlatchDoseTimer".Q )
      Contact( "HMI Tags".AutoRunning )
      Coil( "LatchRPTStart" )
   END_RUNG
   RUNG wire#powerrail
      Contact( "HMI Tags".ModeRepeatTime )
   END_RUNG wire#w1
   RUNG wire#w1
      Contact( "LatchRPTStart" )
   END_RUNG wire#w2
   RUNG wire#powerrail
      Contact( "LatchRPTStart" )
      wire#w3
      Contact( "StopDoseVal" )
      wire#w4
      I_Contact( "UnlatchDoseTimer".Q )
      Coil( "LatchRPTStop" )
   END_RUNG
   RUNG wire#w3
      Contact( "StopDoseTime" )
   END_RUNG wire#w4
   RUNG wire#w3
      Contact( "LatchRPTStop" )
   END_RUNG wire#w4
   RUNG wire#powerrail
      Contact( "LatchRPTStop" )
      { S7_Templates := "time_type := Time" } "RepeatDoseTimer".TON(pt := "HMI Tags".IntervalTime, et => "HMI Tags".DoseWaiting)
      Coil( "RepeatDose" )
   END_RUNG
   RUNG wire#powerrail
      Sub(in1 := "HMI Tags".IntervalTime, in2 := "RepeatDoseTimer".ET, out => "HMI Tags".DoseWaiting)
   END_RUNG
   RUNG wire#powerrail
      Contact( "RepeatDose" )
      Contact( "CMDDose" )
      { S7_Templates := "time_type := Time" } "UnlatchDoseTimer".TON(pt := t#100ms, et =>)
   END_RUNG
   // the same network as SCL:
   "LatchRPTStart" := (("HMI Tags".ModeRepeat AND "HMI Tags".SystemEnables."Flowmeter Fitted") OR "HMI Tags".ModeRepeatTime) AND ("CMDDose" OR "LatchRPTStart") AND NOT "UnlatchDoseTimer".Q AND "HMI Tags".AutoRunning;
   "LatchRPTStop" := "LatchRPTStart" AND ("StopDoseVal" OR "StopDoseTime" OR "LatchRPTStop") AND NOT "UnlatchDoseTimer".Q;
   "RepeatDoseTimer".TON(IN := "LatchRPTStop", PT := "HMI Tags".IntervalTime, ET => "HMI Tags".DoseWaiting);
   "RepeatDose" := "RepeatDoseTimer".Q;
   "HMI Tags".DoseWaiting := "HMI Tags".IntervalTime - "RepeatDoseTimer".ET;
   "UnlatchDoseTimer".TON(IN := "RepeatDose" AND "CMDDose", PT := t#100ms);
END_REGION

REGION Network 14: Buffer Hopper Level Control
   RUNG wire#powerrail
      Contact( "HMI Tags".AutoRunning )
      Contact( "HMI Tags".SystemEnables.BufferValveFitted )
      wire#w1
      Contact( "BufferMinLevelDebounce".Q )
      wire#w2
      I_Contact( "BufferSPLevelDebounce".Q )
      Coil( "OpenIBCValve" )
   END_RUNG
   RUNG wire#w1
      Contact( "OpenIBCValve" )
   END_RUNG wire#w2
   RUNG wire#w1
      { S7_Templates := "SrcType := Real" } LE_Contact(in1 := "HMI Tags".BufferLevel.ScaledSensor, in2 := "HMI Tags".BufferHopperMinLVL)
      { S7_Templates := "time_type := Time" } "BufferMinLevelDebounce".TON(pt := t#5s, et =>)
   END_RUNG
   RUNG wire#w1
      { S7_Templates := "SrcType := Real" } GE_Contact(in1 := "HMI Tags".BufferLevel.ScaledSensor, in2 := "HMI Tags".BufferHopperLVLSP)
      { S7_Templates := "time_type := Time" } "BufferSPLevelDebounce".TON(pt := T#5s, et =>)
   END_RUNG
   // the same network as SCL:
   #_w1 := "HMI Tags".AutoRunning AND "HMI Tags".SystemEnables.BufferValveFitted;
   "OpenIBCValve" := #_w1 AND ("BufferMinLevelDebounce".Q OR "OpenIBCValve") AND NOT "BufferSPLevelDebounce".Q;
   "BufferMinLevelDebounce".TON(IN := #_w1 AND ("HMI Tags".BufferLevel.ScaledSensor <= "HMI Tags".BufferHopperMinLVL),
                           PT := t#5s);
   "BufferSPLevelDebounce".TON(IN := #_w1 AND ("HMI Tags".BufferLevel.ScaledSensor >= "HMI Tags".BufferHopperLVLSP),
                           PT := T#5s);
END_REGION

REGION Network 15: Calc dosing time
   RUNG wire#powerrail
      Contact( "CMDDose" )
      { S7_Templates := "time_type := Time" } "IEC_Timer_0_DB_6".TONR(r := wire#w1, pt := t#120h, et => "HMI Tags".DoseActTime)
   END_RUNG
   RUNG wire#powerrail
      I_Contact( "CMDDose" )
      I_Contact( "StopDoseVal" )
      I_Contact( "StopDoseTime" )
   END_RUNG wire#w1
   // the same network as SCL:
   "IEC_Timer_0_DB_6".TONR(IN := "CMDDose",
                           R := NOT "CMDDose" AND NOT "StopDoseVal" AND NOT "StopDoseTime",
                           PT := t#120h,
                           ET => "HMI Tags".DoseActTime);
END_REGION

REGION Network 16: flowmeter Temperature
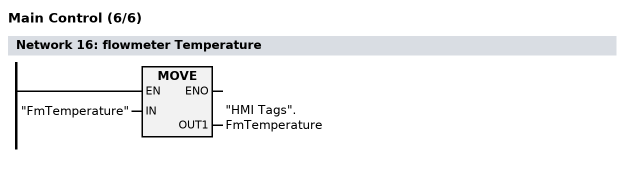
   RUNG wire#powerrail
      Move(in := "FmTemperature", out1 => "HMI Tags".FmTemperature)
   END_RUNG
   // the same network as SCL:
   "HMI Tags".FmTemperature := "FmTemperature";
END_REGION
END_FUNCTION_BLOCK

FUNCTION_BLOCK "FmControl"   // FB6, LAD
{ S7_Optimized_Access := 'TRUE' }
// stored: MemoryReserve 100, SetENOAutomatically false
   VAR_INPUT
      Totalise : Bool;
      "Stop & Reset Count" : Bool;
      "Stop & Preset Value" : Bool;
      "reset and totalise" : Bool;
      "Reset  & Restart" : Bool;
      "Preset and Start" : Bool;
      Hold : Bool;
   END_VAR
   VAR_OUTPUT
      FmTotaliserControl : Byte;
   END_VAR
BEGIN

REGION Network 1: The totalizer is started or continues running.
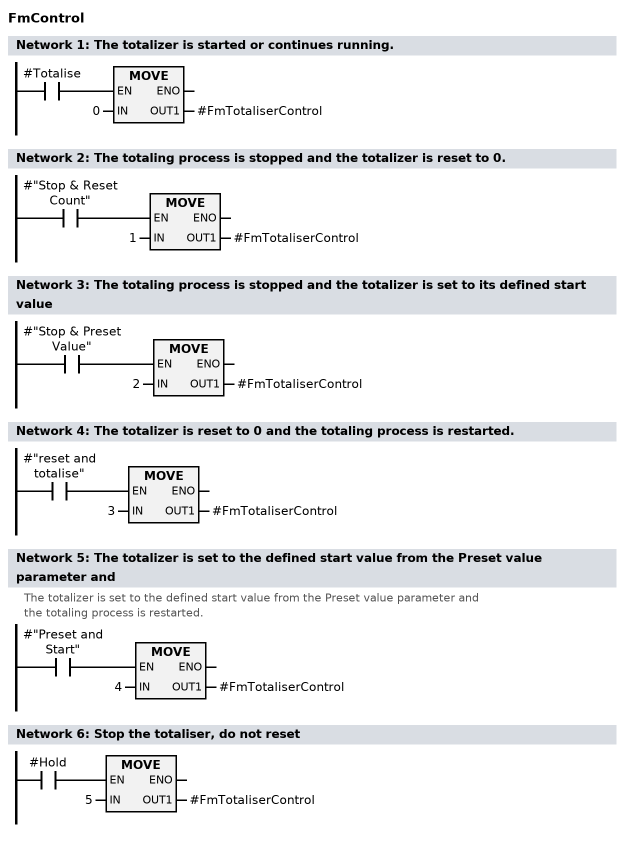
   RUNG wire#powerrail
      Contact( #Totalise )
      Move(in := 0, out1 => #FmTotaliserControl)
   END_RUNG
   // the same network as SCL:
   IF #Totalise THEN #FmTotaliserControl := 0; END_IF;
END_REGION

REGION Network 2: The totaling process is stopped and the totalizer is reset to 0.
   RUNG wire#powerrail
      Contact( #"Stop & Reset Count" )
      Move(in := 1, out1 => #FmTotaliserControl)
   END_RUNG
   // the same network as SCL:
   IF #"Stop & Reset Count" THEN #FmTotaliserControl := 1; END_IF;
END_REGION

REGION Network 3: The totaling process is stopped and the totalizer is set to its defined start value
   RUNG wire#powerrail
      Contact( #"Stop & Preset Value" )
      Move(in := 2, out1 => #FmTotaliserControl)
   END_RUNG
   // the same network as SCL:
   IF #"Stop & Preset Value" THEN #FmTotaliserControl := 2; END_IF;
END_REGION

REGION Network 4: The totalizer is reset to 0 and the totaling process is restarted.
   RUNG wire#powerrail
      Contact( #"reset and totalise" )
      Move(in := 3, out1 => #FmTotaliserControl)
   END_RUNG
   // the same network as SCL:
   IF #"reset and totalise" THEN #FmTotaliserControl := 3; END_IF;
END_REGION

REGION Network 5: The totalizer is set to the defined start value from the Preset value parameter and
   // The totalizer is set to the defined start value from the Preset value parameter and
   // the totaling process is restarted.
   RUNG wire#powerrail
      Contact( #"Preset and Start" )
      Move(in := 4, out1 => #FmTotaliserControl)
   END_RUNG
   // the same network as SCL:
   IF #"Preset and Start" THEN #FmTotaliserControl := 4; END_IF;
END_REGION

REGION Network 6: Stop the totaliser, do not reset
   RUNG wire#powerrail
      Contact( #Hold )
      Move(in := 5, out1 => #FmTotaliserControl)
   END_RUNG
   // the same network as SCL:
   IF #Hold THEN #FmTotaliserControl := 5; END_IF;
END_REGION
END_FUNCTION_BLOCK

FUNCTION "Valve Control" : Void   // FC5, LAD
{ S7_Optimized_Access := 'TRUE' }
// stored: SetENOAutomatically false
BEGIN

REGION Network 1: IBC Valve Control
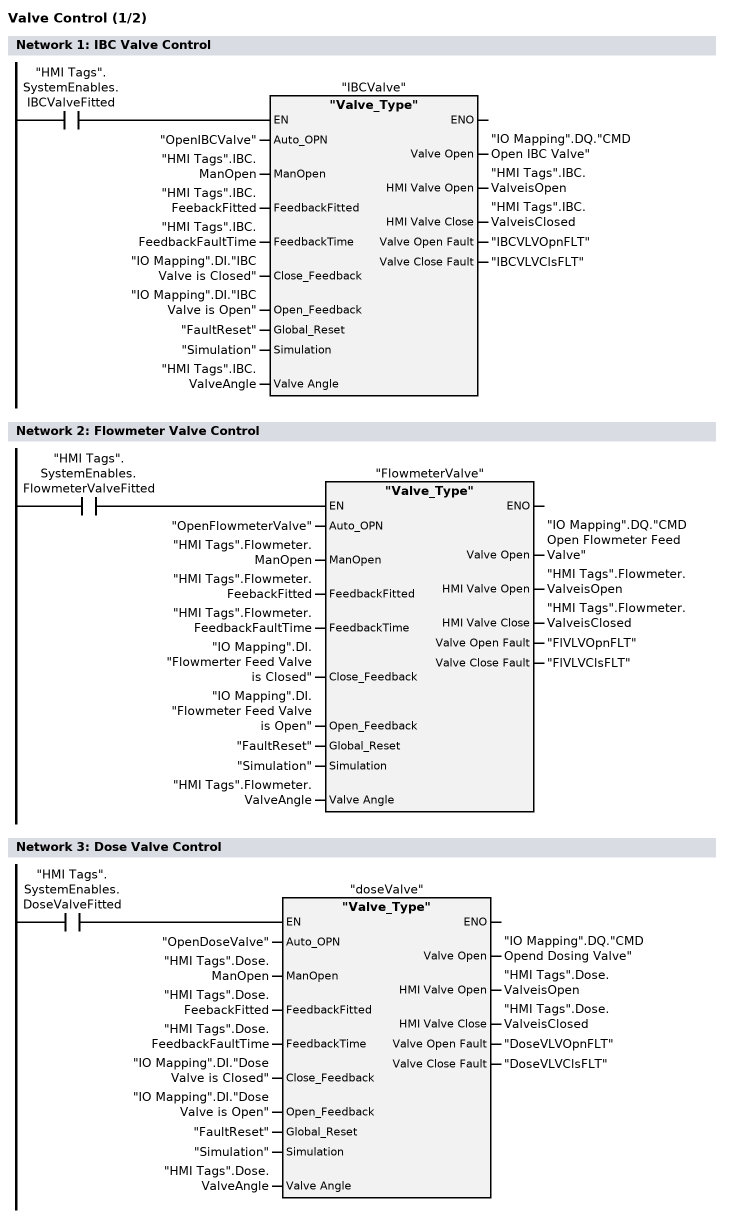
   RUNG wire#powerrail
      Contact( "HMI Tags".SystemEnables.IBCValveFitted )
      "IBCValve"(Auto_OPN := "OpenIBCValve", ManOpen := "HMI Tags".IBC.ManOpen, FeedbackFitted := "HMI Tags".IBC.FeebackFitted, FeedbackTime := "HMI Tags".IBC.FeedbackFaultTime, Close_Feedback := "IO Mapping".DI."IBC Valve is Closed", Open_Feedback := "IO Mapping".DI."IBC Valve is Open", Global_Reset := "FaultReset", Simulation := "Simulation", "Valve Angle" := "HMI Tags".IBC.ValveAngle, "Valve Open" => "IO Mapping".DQ."CMD Open IBC Valve", "HMI Valve Open" => "HMI Tags".IBC.ValveisOpen, "HMI Valve Close" => "HMI Tags".IBC.ValveisClosed, "Valve Open Fault" => "IBCVLVOpnFLT", "Valve Close Fault" => "IBCVLVClsFLT")
   END_RUNG
   // the same network as SCL:
   IF "HMI Tags".SystemEnables.IBCValveFitted THEN
       "IBCValve"(Auto_OPN := "OpenIBCValve",   // "Valve_Type"
                  ManOpen := "HMI Tags".IBC.ManOpen,
                  FeedbackFitted := "HMI Tags".IBC.FeebackFitted,
                  FeedbackTime := "HMI Tags".IBC.FeedbackFaultTime,
                  Close_Feedback := "IO Mapping".DI."IBC Valve is Closed",
                  Open_Feedback := "IO Mapping".DI."IBC Valve is Open",
                  Global_Reset := "FaultReset",
                  Simulation := "Simulation",
                  "Valve Angle" := "HMI Tags".IBC.ValveAngle,
                  "Valve Open" => "IO Mapping".DQ."CMD Open IBC Valve",
                  "HMI Valve Open" => "HMI Tags".IBC.ValveisOpen,
                  "HMI Valve Close" => "HMI Tags".IBC.ValveisClosed,
                  "Valve Open Fault" => "IBCVLVOpnFLT",
                  "Valve Close Fault" => "IBCVLVClsFLT");
   END_IF;
END_REGION

REGION Network 2: Flowmeter Valve Control
   RUNG wire#powerrail
      Contact( "HMI Tags".SystemEnables.FlowmeterValveFitted )
      "FlowmeterValve"(Auto_OPN := "OpenFlowmeterValve", ManOpen := "HMI Tags".Flowmeter.ManOpen, FeedbackFitted := "HMI Tags".Flowmeter.FeebackFitted, FeedbackTime := "HMI Tags".Flowmeter.FeedbackFaultTime, Close_Feedback := "IO Mapping".DI."Flowmerter Feed Valve is Closed", Open_Feedback := "IO Mapping".DI."Flowmeter Feed Valve is Open", Global_Reset := "FaultReset", Simulation := "Simulation", "Valve Angle" := "HMI Tags".Flowmeter.ValveAngle, "Valve Open" => "IO Mapping".DQ."CMD Open Flowmeter Feed Valve", "HMI Valve Open" => "HMI Tags".Flowmeter.ValveisOpen, "HMI Valve Close" => "HMI Tags".Flowmeter.ValveisClosed, "Valve Open Fault" => "FlVLVOpnFLT", "Valve Close Fault" => "FlVLVClsFLT")
   END_RUNG
   // the same network as SCL:
   IF "HMI Tags".SystemEnables.FlowmeterValveFitted THEN
       "FlowmeterValve"(Auto_OPN := "OpenFlowmeterValve",   // "Valve_Type"
                        ManOpen := "HMI Tags".Flowmeter.ManOpen,
                        FeedbackFitted := "HMI Tags".Flowmeter.FeebackFitted,
                        FeedbackTime := "HMI Tags".Flowmeter.FeedbackFaultTime,
                        Close_Feedback := "IO Mapping".DI."Flowmerter Feed Valve is Closed",
                        Open_Feedback := "IO Mapping".DI."Flowmeter Feed Valve is Open",
                        Global_Reset := "FaultReset",
                        Simulation := "Simulation",
                        "Valve Angle" := "HMI Tags".Flowmeter.ValveAngle,
                        "Valve Open" => "IO Mapping".DQ."CMD Open Flowmeter Feed Valve",
                        "HMI Valve Open" => "HMI Tags".Flowmeter.ValveisOpen,
                        "HMI Valve Close" => "HMI Tags".Flowmeter.ValveisClosed,
                        "Valve Open Fault" => "FlVLVOpnFLT",
                        "Valve Close Fault" => "FlVLVClsFLT");
   END_IF;
END_REGION

REGION Network 3: Dose Valve Control
   RUNG wire#powerrail
      Contact( "HMI Tags".SystemEnables.DoseValveFitted )
      "doseValve"(Auto_OPN := "OpenDoseValve", ManOpen := "HMI Tags".Dose.ManOpen, FeedbackFitted := "HMI Tags".Dose.FeebackFitted, FeedbackTime := "HMI Tags".Dose.FeedbackFaultTime, Close_Feedback := "IO Mapping".DI."Dose Valve is Closed", Open_Feedback := "IO Mapping".DI."Dose Valve is Open", Global_Reset := "FaultReset", Simulation := "Simulation", "Valve Angle" := "HMI Tags".Dose.ValveAngle, "Valve Open" => "IO Mapping".DQ."CMD Opend Dosing Valve", "HMI Valve Open" => "HMI Tags".Dose.ValveisOpen, "HMI Valve Close" => "HMI Tags".Dose.ValveisClosed, "Valve Open Fault" => "DoseVLVOpnFLT", "Valve Close Fault" => "DoseVLVClsFLT")
   END_RUNG
   // the same network as SCL:
   IF "HMI Tags".SystemEnables.DoseValveFitted THEN
       "doseValve"(Auto_OPN := "OpenDoseValve",   // "Valve_Type"
                   ManOpen := "HMI Tags".Dose.ManOpen,
                   FeedbackFitted := "HMI Tags".Dose.FeebackFitted,
                   FeedbackTime := "HMI Tags".Dose.FeedbackFaultTime,
                   Close_Feedback := "IO Mapping".DI."Dose Valve is Closed",
                   Open_Feedback := "IO Mapping".DI."Dose Valve is Open",
                   Global_Reset := "FaultReset",
                   Simulation := "Simulation",
                   "Valve Angle" := "HMI Tags".Dose.ValveAngle,
                   "Valve Open" => "IO Mapping".DQ."CMD Opend Dosing Valve",
                   "HMI Valve Open" => "HMI Tags".Dose.ValveisOpen,
                   "HMI Valve Close" => "HMI Tags".Dose.ValveisClosed,
                   "Valve Open Fault" => "DoseVLVOpnFLT",
                   "Valve Close Fault" => "DoseVLVClsFLT");
   END_IF;
END_REGION

REGION Network 4: Pump Valve Control
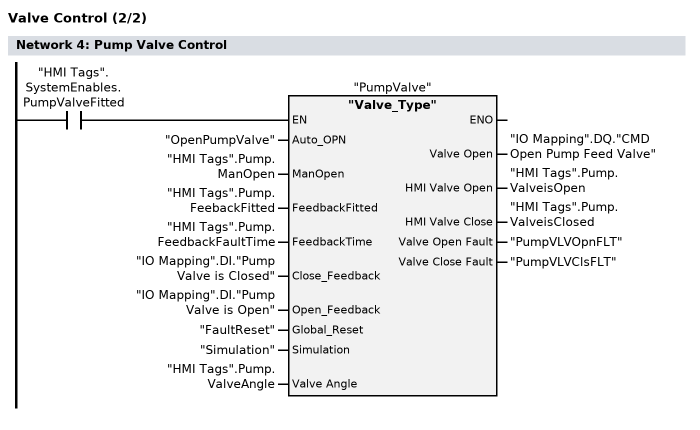
   RUNG wire#powerrail
      Contact( "HMI Tags".SystemEnables.PumpValveFitted )
      "PumpValve"(Auto_OPN := "OpenPumpValve", ManOpen := "HMI Tags".Pump.ManOpen, FeedbackFitted := "HMI Tags".Pump.FeebackFitted, FeedbackTime := "HMI Tags".Pump.FeedbackFaultTime, Close_Feedback := "IO Mapping".DI."Pump Valve is Closed", Open_Feedback := "IO Mapping".DI."Pump Valve is Open", Global_Reset := "FaultReset", Simulation := "Simulation", "Valve Angle" := "HMI Tags".Pump.ValveAngle, "Valve Open" => "IO Mapping".DQ."CMD Open Pump Feed Valve", "HMI Valve Open" => "HMI Tags".Pump.ValveisOpen, "HMI Valve Close" => "HMI Tags".Pump.ValveisClosed, "Valve Open Fault" => "PumpVLVOpnFLT", "Valve Close Fault" => "PumpVLVClsFLT")
   END_RUNG
   // the same network as SCL:
   IF "HMI Tags".SystemEnables.PumpValveFitted THEN
       "PumpValve"(Auto_OPN := "OpenPumpValve",   // "Valve_Type"
                   ManOpen := "HMI Tags".Pump.ManOpen,
                   FeedbackFitted := "HMI Tags".Pump.FeebackFitted,
                   FeedbackTime := "HMI Tags".Pump.FeedbackFaultTime,
                   Close_Feedback := "IO Mapping".DI."Pump Valve is Closed",
                   Open_Feedback := "IO Mapping".DI."Pump Valve is Open",
                   Global_Reset := "FaultReset",
                   Simulation := "Simulation",
                   "Valve Angle" := "HMI Tags".Pump.ValveAngle,
                   "Valve Open" => "IO Mapping".DQ."CMD Open Pump Feed Valve",
                   "HMI Valve Open" => "HMI Tags".Pump.ValveisOpen,
                   "HMI Valve Close" => "HMI Tags".Pump.ValveisClosed,
                   "Valve Open Fault" => "PumpVLVOpnFLT",
                   "Valve Close Fault" => "PumpVLVClsFLT");
   END_IF;
END_REGION
END_FUNCTION

FUNCTION_BLOCK "Valve_Type"   // FB8, LAD
{ S7_Optimized_Access := 'TRUE' }
// stored: MemoryReserve 100, SetENOAutomatically false
   VAR_INPUT
      Auto_OPN : Bool;
      ManOpen : Bool;
      FeedbackFitted : Bool;
      FeedbackTime : Time;
      Close_Feedback : Bool;
      Open_Feedback : Bool;
      Global_Reset : Bool;
      Simulation : Bool;
   END_VAR
   VAR_OUTPUT
      "Valve Open" : Bool;
      "HMI Valve Open" : Bool;
      "HMI Valve Close" : Bool;
      "Valve Open Fault" : Bool;
      "Valve Close Fault" : Bool;
   END_VAR
   VAR_IN_OUT
      "Valve Angle" : Real;
   END_VAR
   VAR
      IEC_Timer_0_Instance { S7_SetPoint := 'True'} : TON_TIME;
      IEC_Timer_0_Instance_1 { S7_SetPoint := 'True'} : TON_TIME;
      "trig 1" : Bool;
      "trig 2" : Bool;
   END_VAR
   VAR_TEMP
      fault_check : Bool;
   END_VAR
   VAR_TEMP   // added for the SCL form of the ladder/FBD networks
      _w1 : Bool;
      _w2 : Bool;
      _w3 : Bool;
      _w4 : Bool;
   END_VAR
BEGIN

REGION Network 1
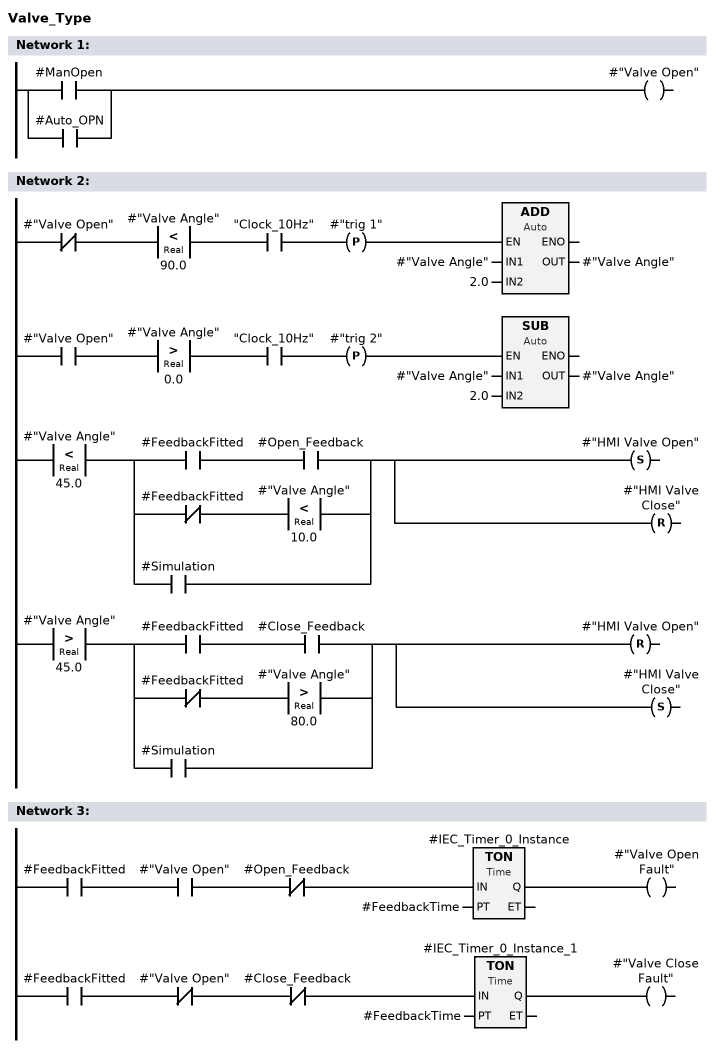
   RUNG wire#powerrail
      Contact( #ManOpen )
      wire#w1
      Coil( #"Valve Open" )
   END_RUNG
   RUNG wire#powerrail
      Contact( #Auto_OPN )
   END_RUNG wire#w1
   // the same network as SCL:
   #"Valve Open" := #ManOpen OR #Auto_OPN;
END_REGION

REGION Network 2
   RUNG wire#powerrail
      I_Contact( #"Valve Open" )
      { S7_Templates := "SrcType := Real" } LT_Contact(in1 := #"Valve Angle", in2 := 90.0)
      Contact( "Clock_10Hz" )
      P_Trig( #"trig 1" )
      Add(in1 := #"Valve Angle", in2 := 2.0, out => #"Valve Angle")
   END_RUNG
   RUNG wire#powerrail
      Contact( #"Valve Open" )
      { S7_Templates := "SrcType := Real" } GT_Contact(in1 := #"Valve Angle", in2 := 0.0)
      Contact( "Clock_10Hz" )
      P_Trig( #"trig 2" )
      Sub(in1 := #"Valve Angle", in2 := 2.0, out => #"Valve Angle")
   END_RUNG
   RUNG wire#powerrail
      { S7_Templates := "SrcType := Real" } LT_Contact(in1 := #"Valve Angle", in2 := 45.0)
      wire#w1
      Contact( #FeedbackFitted )
      Contact( #Open_Feedback )
      wire#w2
      S_Coil( #"HMI Valve Open" )
   END_RUNG
   RUNG wire#w1
      I_Contact( #FeedbackFitted )
      { S7_Templates := "SrcType := Real" } LT_Contact(in1 := #"Valve Angle", in2 := 10.0)
   END_RUNG wire#w2
   RUNG wire#w1
      Contact( #Simulation )
   END_RUNG wire#w2
   RUNG wire#w2
      R_Coil( #"HMI Valve Close" )
   END_RUNG
   RUNG wire#powerrail
      { S7_Templates := "SrcType := Real" } GT_Contact(in1 := #"Valve Angle", in2 := 45.0)
      wire#w3
      Contact( #FeedbackFitted )
      Contact( #Close_Feedback )
      wire#w4
      R_Coil( #"HMI Valve Open" )
   END_RUNG
   RUNG wire#w3
      I_Contact( #FeedbackFitted )
      { S7_Templates := "SrcType := Real" } GT_Contact(in1 := #"Valve Angle", in2 := 80.0)
   END_RUNG wire#w4
   RUNG wire#w3
      Contact( #Simulation )
   END_RUNG wire#w4
   RUNG wire#w4
      S_Coil( #"HMI Valve Close" )
   END_RUNG
   // the same network as SCL:
   #_w1 := NOT #"Valve Open" AND (#"Valve Angle" < 90.0) AND "Clock_10Hz";
   #_w2 := #_w1 AND NOT #"trig 1";   // rising edge
   #"trig 1" := #_w1;
   IF #_w2 THEN #"Valve Angle" := #"Valve Angle" + 2.0; END_IF;
   #_w3 := #"Valve Open" AND (#"Valve Angle" > 0.0) AND "Clock_10Hz";
   #_w4 := #_w3 AND NOT #"trig 2";   // rising edge
   #"trig 2" := #_w3;
   IF #_w4 THEN #"Valve Angle" := #"Valve Angle" - 2.0; END_IF;
   IF (#"Valve Angle" < 45.0) AND ((#FeedbackFitted AND #Open_Feedback) OR (NOT #FeedbackFitted AND (#"Valve Angle" < 10.0)) OR #Simulation) THEN
       #"HMI Valve Open" := TRUE;
       #"HMI Valve Close" := FALSE;
   END_IF;
   IF (#"Valve Angle" > 45.0) AND ((#FeedbackFitted AND #Close_Feedback) OR (NOT #FeedbackFitted AND (#"Valve Angle" > 80.0)) OR #Simulation) THEN
       #"HMI Valve Open" := FALSE;
       #"HMI Valve Close" := TRUE;
   END_IF;
END_REGION

REGION Network 3
   RUNG wire#powerrail
      Contact( #FeedbackFitted )
      Contact( #"Valve Open" )
      I_Contact( #Open_Feedback )
      { S7_Templates := "time_type := Time" } #IEC_Timer_0_Instance.TON(pt := #FeedbackTime, et =>)
      Coil( #"Valve Open Fault" )
   END_RUNG
   RUNG wire#powerrail
      Contact( #FeedbackFitted )
      I_Contact( #"Valve Open" )
      I_Contact( #Close_Feedback )
      { S7_Templates := "time_type := Time" } #IEC_Timer_0_Instance_1.TON(pt := #FeedbackTime, et =>)
      Coil( #"Valve Close Fault" )
   END_RUNG
   // the same network as SCL:
   #IEC_Timer_0_Instance(IN := #FeedbackFitted AND #"Valve Open" AND NOT #Open_Feedback, PT := #FeedbackTime);   // TON
   #"Valve Open Fault" := #IEC_Timer_0_Instance.Q;
   #IEC_Timer_0_Instance_1(IN := #FeedbackFitted AND NOT #"Valve Open" AND NOT #Close_Feedback,   // TON
                           PT := #FeedbackTime);
   #"Valve Close Fault" := #IEC_Timer_0_Instance_1.Q;
END_REGION
END_FUNCTION_BLOCK

FUNCTION "Analog_IN" : Void   // FC3, LAD
{ S7_Optimized_Access := 'TRUE' }
// stored: SetENOAutomatically false
BEGIN

REGION Network 1
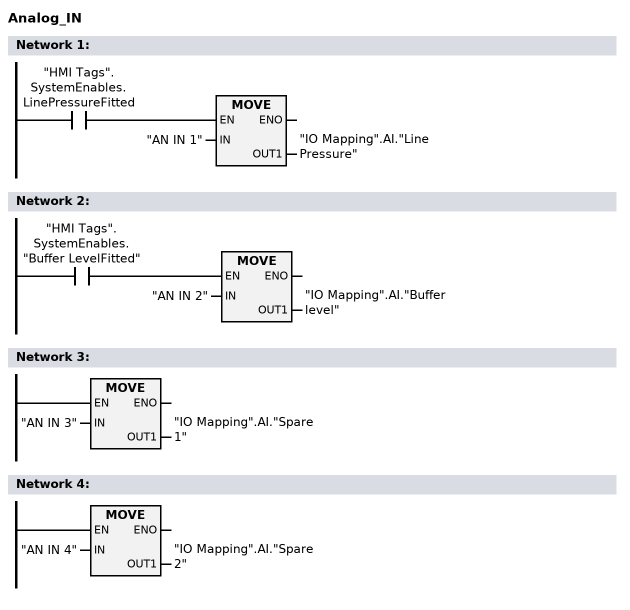
   RUNG wire#powerrail
      Contact( "HMI Tags".SystemEnables.LinePressureFitted )
      Move(in := "AN IN 1", out1 => "IO Mapping".AI."Line Pressure")
   END_RUNG
   // the same network as SCL:
   IF "HMI Tags".SystemEnables.LinePressureFitted THEN "IO Mapping".AI."Line Pressure" := "AN IN 1"; END_IF;
END_REGION

REGION Network 2
   RUNG wire#powerrail
      Contact( "HMI Tags".SystemEnables."Buffer LevelFitted" )
      Move(in := "AN IN 2", out1 => "IO Mapping".AI."Buffer level")
   END_RUNG
   // the same network as SCL:
   IF "HMI Tags".SystemEnables."Buffer LevelFitted" THEN "IO Mapping".AI."Buffer level" := "AN IN 2"; END_IF;
END_REGION

REGION Network 3
   RUNG wire#powerrail
      Move(in := "AN IN 3", out1 => "IO Mapping".AI."Spare 1")
   END_RUNG
   // the same network as SCL:
   "IO Mapping".AI."Spare 1" := "AN IN 3";
END_REGION

REGION Network 4
   RUNG wire#powerrail
      Move(in := "AN IN 4", out1 => "IO Mapping".AI."Spare 2")
   END_RUNG
   // the same network as SCL:
   "IO Mapping".AI."Spare 2" := "AN IN 4";
END_REGION
END_FUNCTION

FUNCTION "Digital_IN" : Void   // FC1, LAD
{ S7_Optimized_Access := 'TRUE' }
// stored: SetENOAutomatically false
BEGIN

REGION Network 1: Safety OK
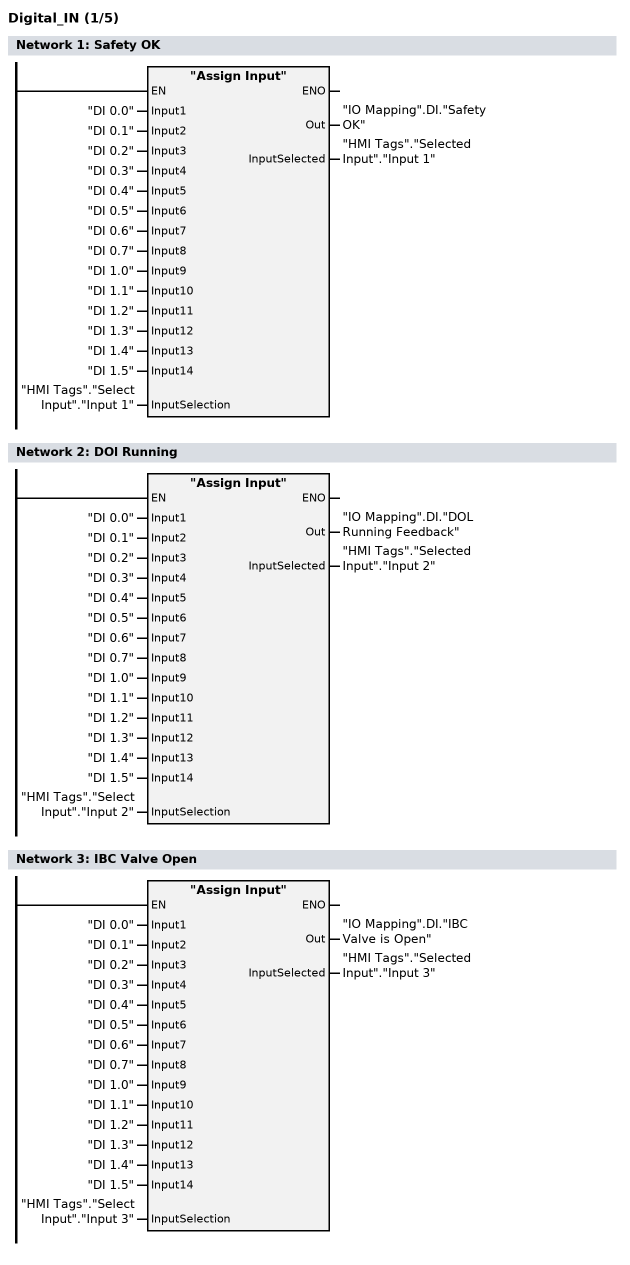
   RUNG wire#powerrail
      "Assign Input"(Input1 := "DI 0.0", Input2 := "DI 0.1", Input3 := "DI 0.2", Input4 := "DI 0.3", Input5 := "DI 0.4", Input6 := "DI 0.5", Input7 := "DI 0.6", Input8 := "DI 0.7", Input9 := "DI 1.0", Input10 := "DI 1.1", Input11 := "DI 1.2", Input12 := "DI 1.3", Input13 := "DI 1.4", Input14 := "DI 1.5", InputSelection := "HMI Tags"."Select Input"."Input 1", Out => "IO Mapping".DI."Safety OK", InputSelected => "HMI Tags"."Selected Input"."Input 1")
   END_RUNG
   // the same network as SCL:
   "Assign Input"(Input1 := "DI 0.0",
                  Input2 := "DI 0.1",
                  Input3 := "DI 0.2",
                  Input4 := "DI 0.3",
                  Input5 := "DI 0.4",
                  Input6 := "DI 0.5",
                  Input7 := "DI 0.6",
                  Input8 := "DI 0.7",
                  Input9 := "DI 1.0",
                  Input10 := "DI 1.1",
                  Input11 := "DI 1.2",
                  Input12 := "DI 1.3",
                  Input13 := "DI 1.4",
                  Input14 := "DI 1.5",
                  InputSelection := "HMI Tags"."Select Input"."Input 1",
                  Out => "IO Mapping".DI."Safety OK",
                  InputSelected => "HMI Tags"."Selected Input"."Input 1");
END_REGION

REGION Network 2: DOl Running
   RUNG wire#powerrail
      "Assign Input"(Input1 := "DI 0.0", Input2 := "DI 0.1", Input3 := "DI 0.2", Input4 := "DI 0.3", Input5 := "DI 0.4", Input6 := "DI 0.5", Input7 := "DI 0.6", Input8 := "DI 0.7", Input9 := "DI 1.0", Input10 := "DI 1.1", Input11 := "DI 1.2", Input12 := "DI 1.3", Input13 := "DI 1.4", Input14 := "DI 1.5", InputSelection := "HMI Tags"."Select Input"."Input 2", Out => "IO Mapping".DI."DOL Running Feedback", InputSelected => "HMI Tags"."Selected Input"."Input 2")
   END_RUNG
   // the same network as SCL:
   "Assign Input"(Input1 := "DI 0.0",
                  Input2 := "DI 0.1",
                  Input3 := "DI 0.2",
                  Input4 := "DI 0.3",
                  Input5 := "DI 0.4",
                  Input6 := "DI 0.5",
                  Input7 := "DI 0.6",
                  Input8 := "DI 0.7",
                  Input9 := "DI 1.0",
                  Input10 := "DI 1.1",
                  Input11 := "DI 1.2",
                  Input12 := "DI 1.3",
                  Input13 := "DI 1.4",
                  Input14 := "DI 1.5",
                  InputSelection := "HMI Tags"."Select Input"."Input 2",
                  Out => "IO Mapping".DI."DOL Running Feedback",
                  InputSelected => "HMI Tags"."Selected Input"."Input 2");
END_REGION

REGION Network 3: IBC Valve Open
   RUNG wire#powerrail
      "Assign Input"(Input1 := "DI 0.0", Input2 := "DI 0.1", Input3 := "DI 0.2", Input4 := "DI 0.3", Input5 := "DI 0.4", Input6 := "DI 0.5", Input7 := "DI 0.6", Input8 := "DI 0.7", Input9 := "DI 1.0", Input10 := "DI 1.1", Input11 := "DI 1.2", Input12 := "DI 1.3", Input13 := "DI 1.4", Input14 := "DI 1.5", InputSelection := "HMI Tags"."Select Input"."Input 3", Out => "IO Mapping".DI."IBC Valve is Open", InputSelected => "HMI Tags"."Selected Input"."Input 3")
   END_RUNG
   // the same network as SCL:
   "Assign Input"(Input1 := "DI 0.0",
                  Input2 := "DI 0.1",
                  Input3 := "DI 0.2",
                  Input4 := "DI 0.3",
                  Input5 := "DI 0.4",
                  Input6 := "DI 0.5",
                  Input7 := "DI 0.6",
                  Input8 := "DI 0.7",
                  Input9 := "DI 1.0",
                  Input10 := "DI 1.1",
                  Input11 := "DI 1.2",
                  Input12 := "DI 1.3",
                  Input13 := "DI 1.4",
                  Input14 := "DI 1.5",
                  InputSelection := "HMI Tags"."Select Input"."Input 3",
                  Out => "IO Mapping".DI."IBC Valve is Open",
                  InputSelected => "HMI Tags"."Selected Input"."Input 3");
END_REGION

REGION Network 4: IBC Valve closed
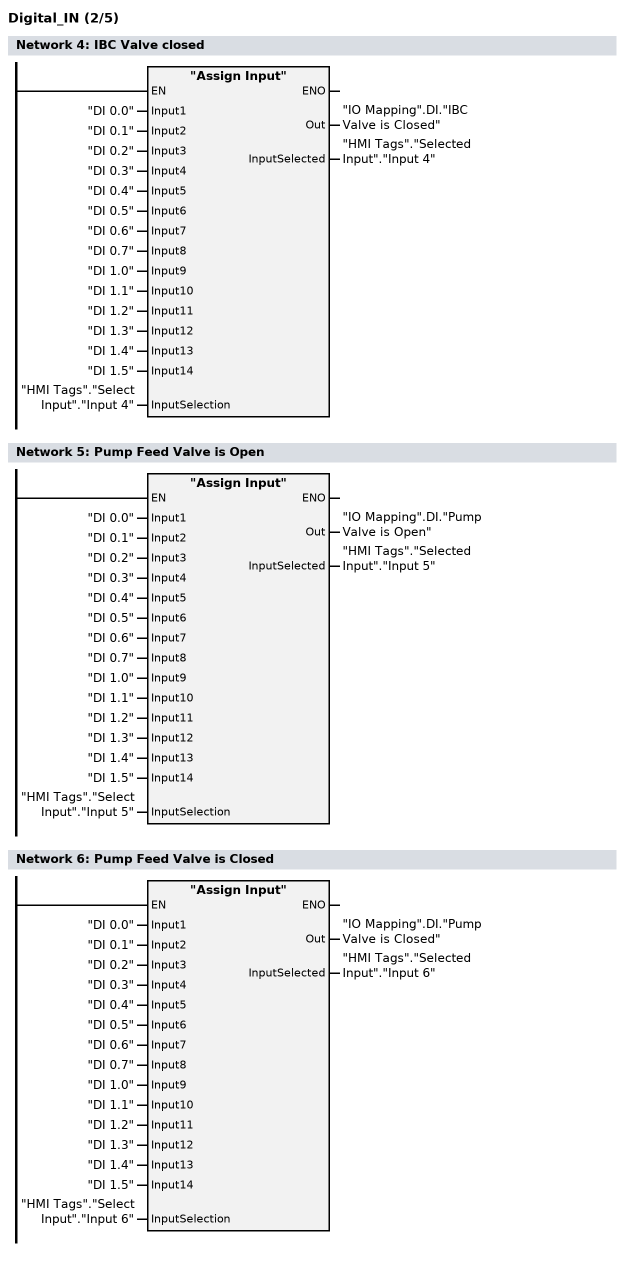
   RUNG wire#powerrail
      "Assign Input"(Input1 := "DI 0.0", Input2 := "DI 0.1", Input3 := "DI 0.2", Input4 := "DI 0.3", Input5 := "DI 0.4", Input6 := "DI 0.5", Input7 := "DI 0.6", Input8 := "DI 0.7", Input9 := "DI 1.0", Input10 := "DI 1.1", Input11 := "DI 1.2", Input12 := "DI 1.3", Input13 := "DI 1.4", Input14 := "DI 1.5", InputSelection := "HMI Tags"."Select Input"."Input 4", Out => "IO Mapping".DI."IBC Valve is Closed", InputSelected => "HMI Tags"."Selected Input"."Input 4")
   END_RUNG
   // the same network as SCL:
   "Assign Input"(Input1 := "DI 0.0",
                  Input2 := "DI 0.1",
                  Input3 := "DI 0.2",
                  Input4 := "DI 0.3",
                  Input5 := "DI 0.4",
                  Input6 := "DI 0.5",
                  Input7 := "DI 0.6",
                  Input8 := "DI 0.7",
                  Input9 := "DI 1.0",
                  Input10 := "DI 1.1",
                  Input11 := "DI 1.2",
                  Input12 := "DI 1.3",
                  Input13 := "DI 1.4",
                  Input14 := "DI 1.5",
                  InputSelection := "HMI Tags"."Select Input"."Input 4",
                  Out => "IO Mapping".DI."IBC Valve is Closed",
                  InputSelected => "HMI Tags"."Selected Input"."Input 4");
END_REGION

REGION Network 5: Pump Feed Valve is Open
   RUNG wire#powerrail
      "Assign Input"(Input1 := "DI 0.0", Input2 := "DI 0.1", Input3 := "DI 0.2", Input4 := "DI 0.3", Input5 := "DI 0.4", Input6 := "DI 0.5", Input7 := "DI 0.6", Input8 := "DI 0.7", Input9 := "DI 1.0", Input10 := "DI 1.1", Input11 := "DI 1.2", Input12 := "DI 1.3", Input13 := "DI 1.4", Input14 := "DI 1.5", InputSelection := "HMI Tags"."Select Input"."Input 5", Out => "IO Mapping".DI."Pump Valve is Open", InputSelected => "HMI Tags"."Selected Input"."Input 5")
   END_RUNG
   // the same network as SCL:
   "Assign Input"(Input1 := "DI 0.0",
                  Input2 := "DI 0.1",
                  Input3 := "DI 0.2",
                  Input4 := "DI 0.3",
                  Input5 := "DI 0.4",
                  Input6 := "DI 0.5",
                  Input7 := "DI 0.6",
                  Input8 := "DI 0.7",
                  Input9 := "DI 1.0",
                  Input10 := "DI 1.1",
                  Input11 := "DI 1.2",
                  Input12 := "DI 1.3",
                  Input13 := "DI 1.4",
                  Input14 := "DI 1.5",
                  InputSelection := "HMI Tags"."Select Input"."Input 5",
                  Out => "IO Mapping".DI."Pump Valve is Open",
                  InputSelected => "HMI Tags"."Selected Input"."Input 5");
END_REGION

REGION Network 6: Pump Feed Valve is Closed
   RUNG wire#powerrail
      "Assign Input"(Input1 := "DI 0.0", Input2 := "DI 0.1", Input3 := "DI 0.2", Input4 := "DI 0.3", Input5 := "DI 0.4", Input6 := "DI 0.5", Input7 := "DI 0.6", Input8 := "DI 0.7", Input9 := "DI 1.0", Input10 := "DI 1.1", Input11 := "DI 1.2", Input12 := "DI 1.3", Input13 := "DI 1.4", Input14 := "DI 1.5", InputSelection := "HMI Tags"."Select Input"."Input 6", Out => "IO Mapping".DI."Pump Valve is Closed", InputSelected => "HMI Tags"."Selected Input"."Input 6")
   END_RUNG
   // the same network as SCL:
   "Assign Input"(Input1 := "DI 0.0",
                  Input2 := "DI 0.1",
                  Input3 := "DI 0.2",
                  Input4 := "DI 0.3",
                  Input5 := "DI 0.4",
                  Input6 := "DI 0.5",
                  Input7 := "DI 0.6",
                  Input8 := "DI 0.7",
                  Input9 := "DI 1.0",
                  Input10 := "DI 1.1",
                  Input11 := "DI 1.2",
                  Input12 := "DI 1.3",
                  Input13 := "DI 1.4",
                  Input14 := "DI 1.5",
                  InputSelection := "HMI Tags"."Select Input"."Input 6",
                  Out => "IO Mapping".DI."Pump Valve is Closed",
                  InputSelected => "HMI Tags"."Selected Input"."Input 6");
END_REGION

REGION Network 7: Flometer Feed Valve is Open
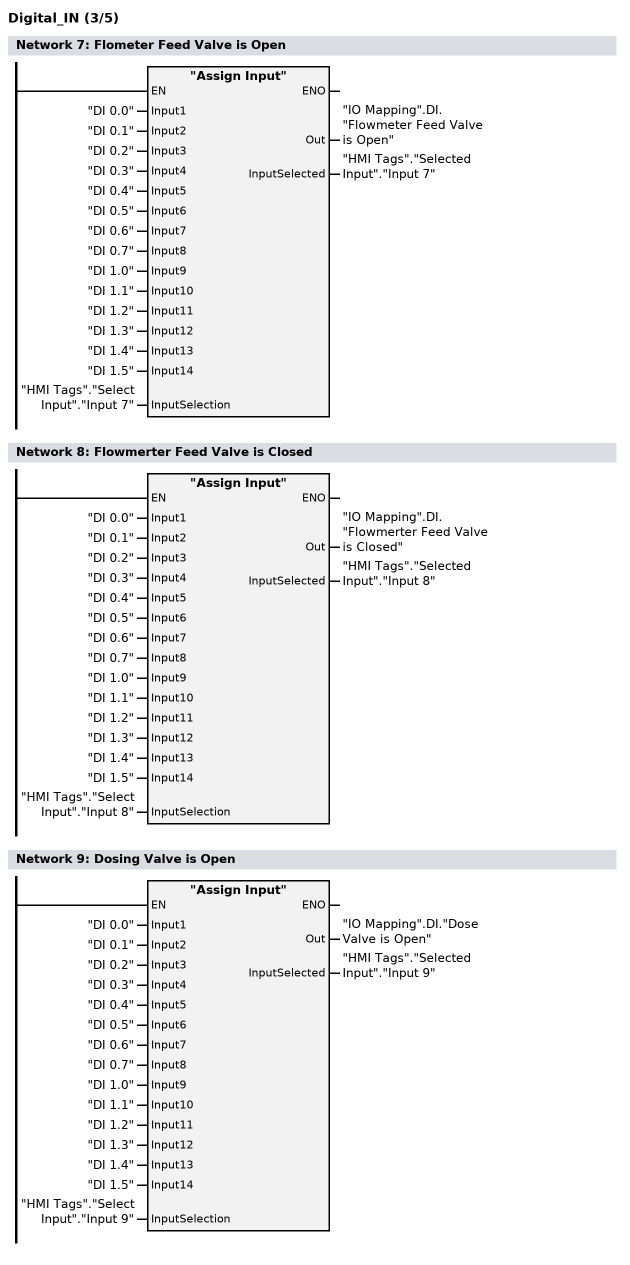
   RUNG wire#powerrail
      "Assign Input"(Input1 := "DI 0.0", Input2 := "DI 0.1", Input3 := "DI 0.2", Input4 := "DI 0.3", Input5 := "DI 0.4", Input6 := "DI 0.5", Input7 := "DI 0.6", Input8 := "DI 0.7", Input9 := "DI 1.0", Input10 := "DI 1.1", Input11 := "DI 1.2", Input12 := "DI 1.3", Input13 := "DI 1.4", Input14 := "DI 1.5", InputSelection := "HMI Tags"."Select Input"."Input 7", Out => "IO Mapping".DI."Flowmeter Feed Valve is Open", InputSelected => "HMI Tags"."Selected Input"."Input 7")
   END_RUNG
   // the same network as SCL:
   "Assign Input"(Input1 := "DI 0.0",
                  Input2 := "DI 0.1",
                  Input3 := "DI 0.2",
                  Input4 := "DI 0.3",
                  Input5 := "DI 0.4",
                  Input6 := "DI 0.5",
                  Input7 := "DI 0.6",
                  Input8 := "DI 0.7",
                  Input9 := "DI 1.0",
                  Input10 := "DI 1.1",
                  Input11 := "DI 1.2",
                  Input12 := "DI 1.3",
                  Input13 := "DI 1.4",
                  Input14 := "DI 1.5",
                  InputSelection := "HMI Tags"."Select Input"."Input 7",
                  Out => "IO Mapping".DI."Flowmeter Feed Valve is Open",
                  InputSelected => "HMI Tags"."Selected Input"."Input 7");
END_REGION

REGION Network 8: Flowmerter Feed Valve is Closed
   RUNG wire#powerrail
      "Assign Input"(Input1 := "DI 0.0", Input2 := "DI 0.1", Input3 := "DI 0.2", Input4 := "DI 0.3", Input5 := "DI 0.4", Input6 := "DI 0.5", Input7 := "DI 0.6", Input8 := "DI 0.7", Input9 := "DI 1.0", Input10 := "DI 1.1", Input11 := "DI 1.2", Input12 := "DI 1.3", Input13 := "DI 1.4", Input14 := "DI 1.5", InputSelection := "HMI Tags"."Select Input"."Input 8", Out => "IO Mapping".DI."Flowmerter Feed Valve is Closed", InputSelected => "HMI Tags"."Selected Input"."Input 8")
   END_RUNG
   // the same network as SCL:
   "Assign Input"(Input1 := "DI 0.0",
                  Input2 := "DI 0.1",
                  Input3 := "DI 0.2",
                  Input4 := "DI 0.3",
                  Input5 := "DI 0.4",
                  Input6 := "DI 0.5",
                  Input7 := "DI 0.6",
                  Input8 := "DI 0.7",
                  Input9 := "DI 1.0",
                  Input10 := "DI 1.1",
                  Input11 := "DI 1.2",
                  Input12 := "DI 1.3",
                  Input13 := "DI 1.4",
                  Input14 := "DI 1.5",
                  InputSelection := "HMI Tags"."Select Input"."Input 8",
                  Out => "IO Mapping".DI."Flowmerter Feed Valve is Closed",
                  InputSelected => "HMI Tags"."Selected Input"."Input 8");
END_REGION

REGION Network 9: Dosing Valve is Open
   RUNG wire#powerrail
      "Assign Input"(Input1 := "DI 0.0", Input2 := "DI 0.1", Input3 := "DI 0.2", Input4 := "DI 0.3", Input5 := "DI 0.4", Input6 := "DI 0.5", Input7 := "DI 0.6", Input8 := "DI 0.7", Input9 := "DI 1.0", Input10 := "DI 1.1", Input11 := "DI 1.2", Input12 := "DI 1.3", Input13 := "DI 1.4", Input14 := "DI 1.5", InputSelection := "HMI Tags"."Select Input"."Input 9", Out => "IO Mapping".DI."Dose Valve is Open", InputSelected => "HMI Tags"."Selected Input"."Input 9")
   END_RUNG
   // the same network as SCL:
   "Assign Input"(Input1 := "DI 0.0",
                  Input2 := "DI 0.1",
                  Input3 := "DI 0.2",
                  Input4 := "DI 0.3",
                  Input5 := "DI 0.4",
                  Input6 := "DI 0.5",
                  Input7 := "DI 0.6",
                  Input8 := "DI 0.7",
                  Input9 := "DI 1.0",
                  Input10 := "DI 1.1",
                  Input11 := "DI 1.2",
                  Input12 := "DI 1.3",
                  Input13 := "DI 1.4",
                  Input14 := "DI 1.5",
                  InputSelection := "HMI Tags"."Select Input"."Input 9",
                  Out => "IO Mapping".DI."Dose Valve is Open",
                  InputSelected => "HMI Tags"."Selected Input"."Input 9");
END_REGION

REGION Network 10: Dosing Valve is Closed
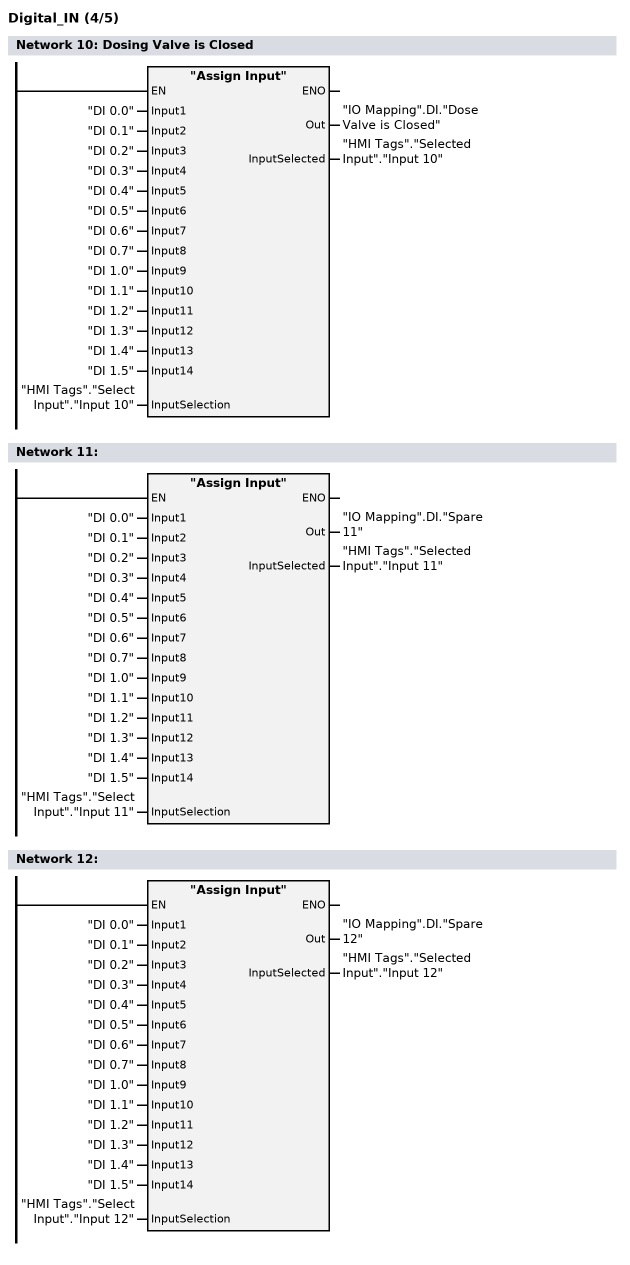
   RUNG wire#powerrail
      "Assign Input"(Input1 := "DI 0.0", Input2 := "DI 0.1", Input3 := "DI 0.2", Input4 := "DI 0.3", Input5 := "DI 0.4", Input6 := "DI 0.5", Input7 := "DI 0.6", Input8 := "DI 0.7", Input9 := "DI 1.0", Input10 := "DI 1.1", Input11 := "DI 1.2", Input12 := "DI 1.3", Input13 := "DI 1.4", Input14 := "DI 1.5", InputSelection := "HMI Tags"."Select Input"."Input 10", Out => "IO Mapping".DI."Dose Valve is Closed", InputSelected => "HMI Tags"."Selected Input"."Input 10")
   END_RUNG
   // the same network as SCL:
   "Assign Input"(Input1 := "DI 0.0",
                  Input2 := "DI 0.1",
                  Input3 := "DI 0.2",
                  Input4 := "DI 0.3",
                  Input5 := "DI 0.4",
                  Input6 := "DI 0.5",
                  Input7 := "DI 0.6",
                  Input8 := "DI 0.7",
                  Input9 := "DI 1.0",
                  Input10 := "DI 1.1",
                  Input11 := "DI 1.2",
                  Input12 := "DI 1.3",
                  Input13 := "DI 1.4",
                  Input14 := "DI 1.5",
                  InputSelection := "HMI Tags"."Select Input"."Input 10",
                  Out => "IO Mapping".DI."Dose Valve is Closed",
                  InputSelected => "HMI Tags"."Selected Input"."Input 10");
END_REGION

REGION Network 11
   RUNG wire#powerrail
      "Assign Input"(Input1 := "DI 0.0", Input2 := "DI 0.1", Input3 := "DI 0.2", Input4 := "DI 0.3", Input5 := "DI 0.4", Input6 := "DI 0.5", Input7 := "DI 0.6", Input8 := "DI 0.7", Input9 := "DI 1.0", Input10 := "DI 1.1", Input11 := "DI 1.2", Input12 := "DI 1.3", Input13 := "DI 1.4", Input14 := "DI 1.5", InputSelection := "HMI Tags"."Select Input"."Input 11", Out => "IO Mapping".DI."Spare 11", InputSelected => "HMI Tags"."Selected Input"."Input 11")
   END_RUNG
   // the same network as SCL:
   "Assign Input"(Input1 := "DI 0.0",
                  Input2 := "DI 0.1",
                  Input3 := "DI 0.2",
                  Input4 := "DI 0.3",
                  Input5 := "DI 0.4",
                  Input6 := "DI 0.5",
                  Input7 := "DI 0.6",
                  Input8 := "DI 0.7",
                  Input9 := "DI 1.0",
                  Input10 := "DI 1.1",
                  Input11 := "DI 1.2",
                  Input12 := "DI 1.3",
                  Input13 := "DI 1.4",
                  Input14 := "DI 1.5",
                  InputSelection := "HMI Tags"."Select Input"."Input 11",
                  Out => "IO Mapping".DI."Spare 11",
                  InputSelected => "HMI Tags"."Selected Input"."Input 11");
END_REGION

REGION Network 12
   RUNG wire#powerrail
      "Assign Input"(Input1 := "DI 0.0", Input2 := "DI 0.1", Input3 := "DI 0.2", Input4 := "DI 0.3", Input5 := "DI 0.4", Input6 := "DI 0.5", Input7 := "DI 0.6", Input8 := "DI 0.7", Input9 := "DI 1.0", Input10 := "DI 1.1", Input11 := "DI 1.2", Input12 := "DI 1.3", Input13 := "DI 1.4", Input14 := "DI 1.5", InputSelection := "HMI Tags"."Select Input"."Input 12", Out => "IO Mapping".DI."Spare 12", InputSelected => "HMI Tags"."Selected Input"."Input 12")
   END_RUNG
   // the same network as SCL:
   "Assign Input"(Input1 := "DI 0.0",
                  Input2 := "DI 0.1",
                  Input3 := "DI 0.2",
                  Input4 := "DI 0.3",
                  Input5 := "DI 0.4",
                  Input6 := "DI 0.5",
                  Input7 := "DI 0.6",
                  Input8 := "DI 0.7",
                  Input9 := "DI 1.0",
                  Input10 := "DI 1.1",
                  Input11 := "DI 1.2",
                  Input12 := "DI 1.3",
                  Input13 := "DI 1.4",
                  Input14 := "DI 1.5",
                  InputSelection := "HMI Tags"."Select Input"."Input 12",
                  Out => "IO Mapping".DI."Spare 12",
                  InputSelected => "HMI Tags"."Selected Input"."Input 12");
END_REGION

REGION Network 13
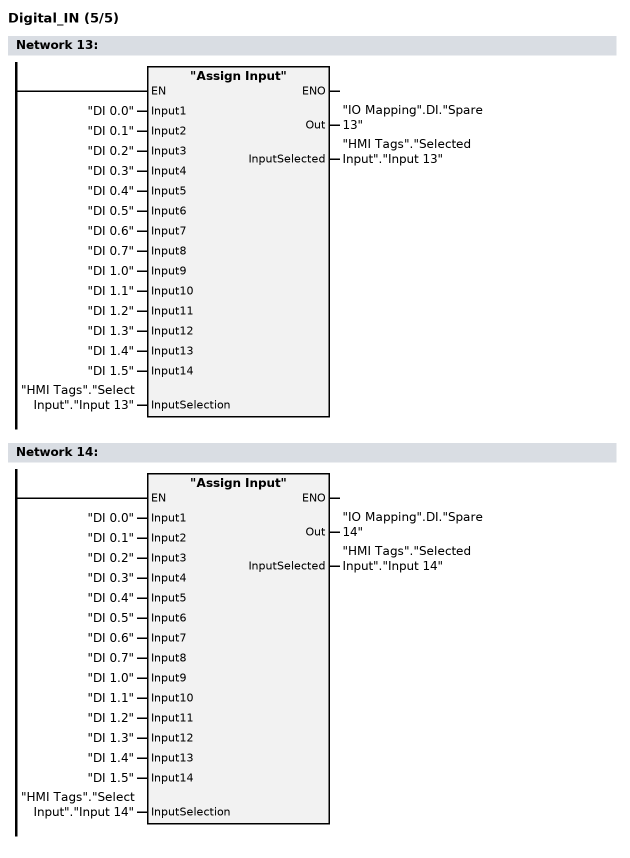
   RUNG wire#powerrail
      "Assign Input"(Input1 := "DI 0.0", Input2 := "DI 0.1", Input3 := "DI 0.2", Input4 := "DI 0.3", Input5 := "DI 0.4", Input6 := "DI 0.5", Input7 := "DI 0.6", Input8 := "DI 0.7", Input9 := "DI 1.0", Input10 := "DI 1.1", Input11 := "DI 1.2", Input12 := "DI 1.3", Input13 := "DI 1.4", Input14 := "DI 1.5", InputSelection := "HMI Tags"."Select Input"."Input 13", Out => "IO Mapping".DI."Spare 13", InputSelected => "HMI Tags"."Selected Input"."Input 13")
   END_RUNG
   // the same network as SCL:
   "Assign Input"(Input1 := "DI 0.0",
                  Input2 := "DI 0.1",
                  Input3 := "DI 0.2",
                  Input4 := "DI 0.3",
                  Input5 := "DI 0.4",
                  Input6 := "DI 0.5",
                  Input7 := "DI 0.6",
                  Input8 := "DI 0.7",
                  Input9 := "DI 1.0",
                  Input10 := "DI 1.1",
                  Input11 := "DI 1.2",
                  Input12 := "DI 1.3",
                  Input13 := "DI 1.4",
                  Input14 := "DI 1.5",
                  InputSelection := "HMI Tags"."Select Input"."Input 13",
                  Out => "IO Mapping".DI."Spare 13",
                  InputSelected => "HMI Tags"."Selected Input"."Input 13");
END_REGION

REGION Network 14
   RUNG wire#powerrail
      "Assign Input"(Input1 := "DI 0.0", Input2 := "DI 0.1", Input3 := "DI 0.2", Input4 := "DI 0.3", Input5 := "DI 0.4", Input6 := "DI 0.5", Input7 := "DI 0.6", Input8 := "DI 0.7", Input9 := "DI 1.0", Input10 := "DI 1.1", Input11 := "DI 1.2", Input12 := "DI 1.3", Input13 := "DI 1.4", Input14 := "DI 1.5", InputSelection := "HMI Tags"."Select Input"."Input 14", Out => "IO Mapping".DI."Spare 14", InputSelected => "HMI Tags"."Selected Input"."Input 14")
   END_RUNG
   // the same network as SCL:
   "Assign Input"(Input1 := "DI 0.0",
                  Input2 := "DI 0.1",
                  Input3 := "DI 0.2",
                  Input4 := "DI 0.3",
                  Input5 := "DI 0.4",
                  Input6 := "DI 0.5",
                  Input7 := "DI 0.6",
                  Input8 := "DI 0.7",
                  Input9 := "DI 1.0",
                  Input10 := "DI 1.1",
                  Input11 := "DI 1.2",
                  Input12 := "DI 1.3",
                  Input13 := "DI 1.4",
                  Input14 := "DI 1.5",
                  InputSelection := "HMI Tags"."Select Input"."Input 14",
                  Out => "IO Mapping".DI."Spare 14",
                  InputSelected => "HMI Tags"."Selected Input"."Input 14");
END_REGION
END_FUNCTION

FUNCTION "Assign Input" : Void   // FC4, LAD
{ S7_Optimized_Access := 'TRUE' }
// stored: SetENOAutomatically false
   VAR_INPUT
      Input1 : Bool;
      Input2 : Bool;
      Input3 : Bool;
      Input4 : Bool;
      Input5 : Bool;
      Input6 : Bool;
      Input7 : Bool;
      Input8 : Bool;
      Input9 : Bool;
      Input10 : Bool;
      Input11 : Bool;
      Input12 : Bool;
      Input13 : Bool;
      Input14 : Bool;
      InputSelection : Int;
   END_VAR
   VAR_OUTPUT
      Out : Bool;
      InputSelected : Int;
   END_VAR
BEGIN

REGION Network 1
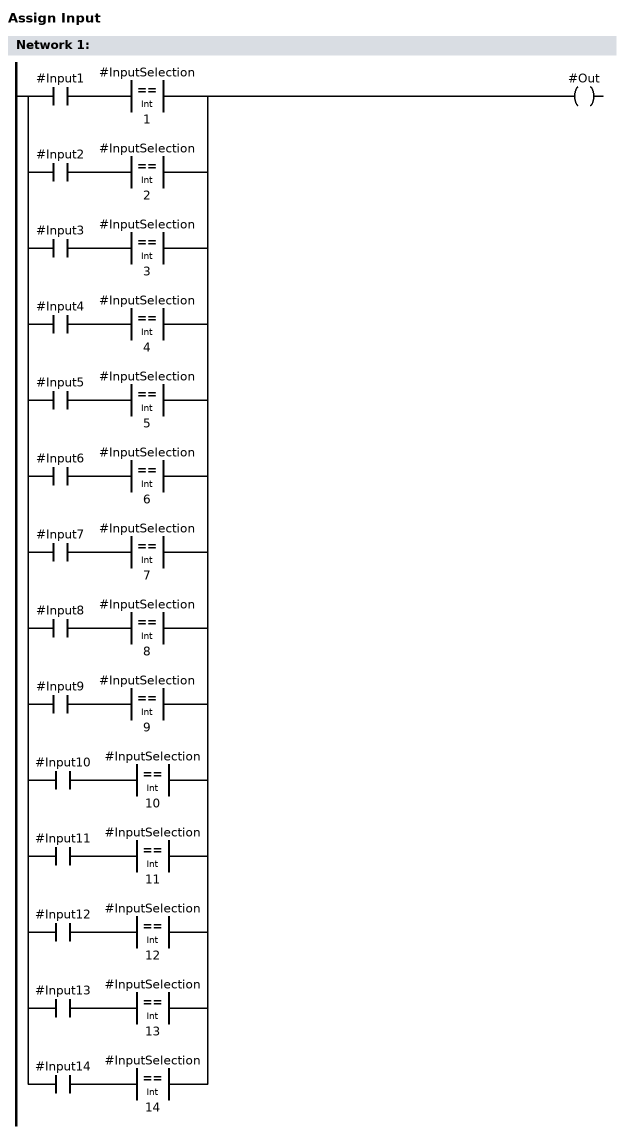
   RUNG wire#powerrail
      Contact( #Input1 )
      { S7_Templates := "SrcType := Int" } EQ_Contact(in1 := #InputSelection, in2 := 1)
      wire#w1
      Coil( #Out )
   END_RUNG
   RUNG wire#powerrail
      Contact( #Input2 )
      { S7_Templates := "SrcType := Int" } EQ_Contact(in1 := #InputSelection, in2 := 2)
   END_RUNG wire#w1
   RUNG wire#powerrail
      Contact( #Input3 )
      { S7_Templates := "SrcType := Int" } EQ_Contact(in1 := #InputSelection, in2 := 3)
   END_RUNG wire#w1
   RUNG wire#powerrail
      Contact( #Input4 )
      { S7_Templates := "SrcType := Int" } EQ_Contact(in1 := #InputSelection, in2 := 4)
   END_RUNG wire#w1
   RUNG wire#powerrail
      Contact( #Input5 )
      { S7_Templates := "SrcType := Int" } EQ_Contact(in1 := #InputSelection, in2 := 5)
   END_RUNG wire#w1
   RUNG wire#powerrail
      Contact( #Input6 )
      { S7_Templates := "SrcType := Int" } EQ_Contact(in1 := #InputSelection, in2 := 6)
   END_RUNG wire#w1
   RUNG wire#powerrail
      Contact( #Input7 )
      { S7_Templates := "SrcType := Int" } EQ_Contact(in1 := #InputSelection, in2 := 7)
   END_RUNG wire#w1
   RUNG wire#powerrail
      Contact( #Input8 )
      { S7_Templates := "SrcType := Int" } EQ_Contact(in1 := #InputSelection, in2 := 8)
   END_RUNG wire#w1
   RUNG wire#powerrail
      Contact( #Input9 )
      { S7_Templates := "SrcType := Int" } EQ_Contact(in1 := #InputSelection, in2 := 9)
   END_RUNG wire#w1
   RUNG wire#powerrail
      Contact( #Input10 )
      { S7_Templates := "SrcType := Int" } EQ_Contact(in1 := #InputSelection, in2 := 10)
   END_RUNG wire#w1
   RUNG wire#powerrail
      Contact( #Input11 )
      { S7_Templates := "SrcType := Int" } EQ_Contact(in1 := #InputSelection, in2 := 11)
   END_RUNG wire#w1
   RUNG wire#powerrail
      Contact( #Input12 )
      { S7_Templates := "SrcType := Int" } EQ_Contact(in1 := #InputSelection, in2 := 12)
   END_RUNG wire#w1
   RUNG wire#powerrail
      Contact( #Input13 )
      { S7_Templates := "SrcType := Int" } EQ_Contact(in1 := #InputSelection, in2 := 13)
   END_RUNG wire#w1
   RUNG wire#powerrail
      Contact( #Input14 )
      { S7_Templates := "SrcType := Int" } EQ_Contact(in1 := #InputSelection, in2 := 14)
   END_RUNG wire#w1
   // the same network as SCL:
   #Out := (#Input1 AND (#InputSelection = 1)) OR (#Input2 AND (#InputSelection = 2)) OR (#Input3 AND (#InputSelection = 3)) OR (#Input4 AND (#InputSelection = 4)) OR (#Input5 AND (#InputSelection = 5)) OR (#Input6 AND (#InputSelection = 6)) OR (#Input7 AND (#InputSelection = 7)) OR (#Input8 AND (#InputSelection = 8)) OR (#Input9 AND (#InputSelection = 9)) OR (#Input10 AND (#InputSelection = 10)) OR (#Input11 AND (#InputSelection = 11)) OR (#Input12 AND (#InputSelection = 12)) OR (#Input13 AND (#InputSelection = 13)) OR (#Input14 AND (#InputSelection = 14));
END_REGION
END_FUNCTION

FUNCTION "Digital_OUT" : Void   // FC2, LAD
{ S7_Optimized_Access := 'TRUE' }
// stored: SetENOAutomatically false
BEGIN

REGION Network 1: CMD Open IBC Valve
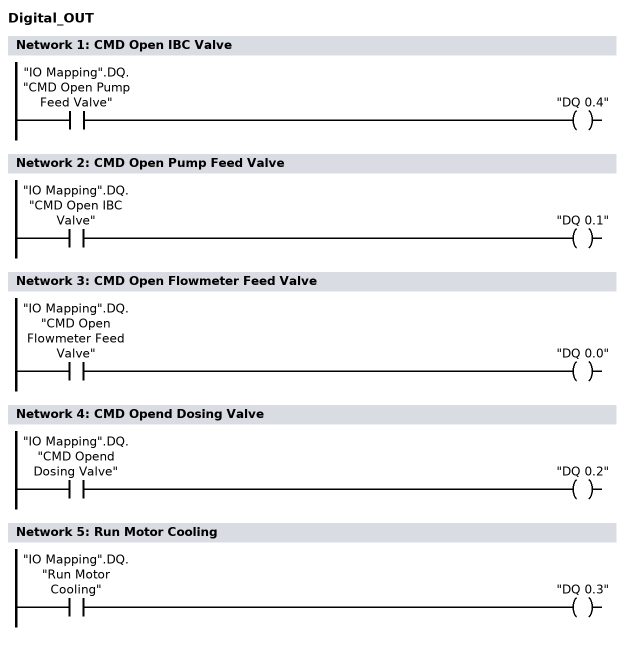
   RUNG wire#powerrail
      Contact( "IO Mapping".DQ."CMD Open Pump Feed Valve" )
      Coil( "DQ 0.4" )
   END_RUNG
   // the same network as SCL:
   "DQ 0.4" := "IO Mapping".DQ."CMD Open Pump Feed Valve";
END_REGION

REGION Network 2: CMD Open Pump Feed Valve
   RUNG wire#powerrail
      Contact( "IO Mapping".DQ."CMD Open IBC Valve" )
      Coil( "DQ 0.1" )
   END_RUNG
   // the same network as SCL:
   "DQ 0.1" := "IO Mapping".DQ."CMD Open IBC Valve";
END_REGION

REGION Network 3: CMD Open Flowmeter Feed Valve
   RUNG wire#powerrail
      Contact( "IO Mapping".DQ."CMD Open Flowmeter Feed Valve" )
      Coil( "DQ 0.0" )
   END_RUNG
   // the same network as SCL:
   "DQ 0.0" := "IO Mapping".DQ."CMD Open Flowmeter Feed Valve";
END_REGION

REGION Network 4: CMD Opend Dosing Valve
   RUNG wire#powerrail
      Contact( "IO Mapping".DQ."CMD Opend Dosing Valve" )
      Coil( "DQ 0.2" )
   END_RUNG
   // the same network as SCL:
   "DQ 0.2" := "IO Mapping".DQ."CMD Opend Dosing Valve";
END_REGION

REGION Network 5: Run Motor Cooling
   RUNG wire#powerrail
      Contact( "IO Mapping".DQ."Run Motor Cooling" )
      Coil( "DQ 0.3" )
   END_RUNG
   // the same network as SCL:
   "DQ 0.3" := "IO Mapping".DQ."Run Motor Cooling";
END_REGION
END_FUNCTION

FUNCTION "DOL Control" : Void   // FC8, LAD
{ S7_Optimized_Access := 'TRUE' }
// stored: SetENOAutomatically false
   VAR_TEMP   // added for the SCL form of the ladder/FBD networks
      _w1 : Bool;
   END_VAR
BEGIN

REGION Network 1: Request Cooling Motor Run
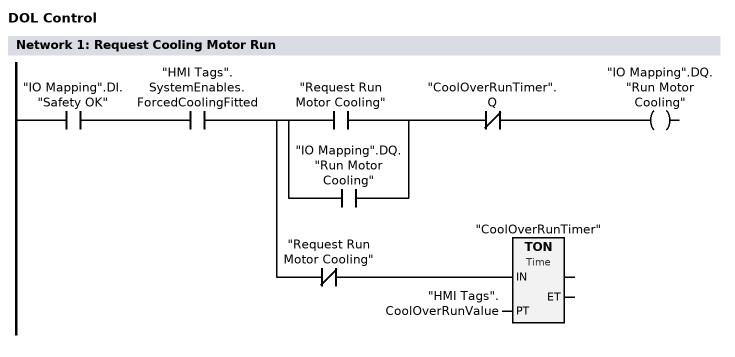
   RUNG wire#powerrail
      Contact( "IO Mapping".DI."Safety OK" )
      Contact( "HMI Tags".SystemEnables.ForcedCoolingFitted )
      wire#w1
      Contact( "Request Run Motor Cooling" )
      wire#w2
      I_Contact( "CoolOverRunTimer".Q )
      Coil( "IO Mapping".DQ."Run Motor Cooling" )
   END_RUNG
   RUNG wire#w1
      Contact( "IO Mapping".DQ."Run Motor Cooling" )
   END_RUNG wire#w2
   RUNG wire#w1
      I_Contact( "Request Run Motor Cooling" )
      { S7_Templates := "time_type := Time" } "CoolOverRunTimer".TON(pt := "HMI Tags".CoolOverRunValue, et =>)
   END_RUNG
   // the same network as SCL:
   #_w1 := "IO Mapping".DI."Safety OK" AND "HMI Tags".SystemEnables.ForcedCoolingFitted;
   "IO Mapping".DQ."Run Motor Cooling" := #_w1 AND ("Request Run Motor Cooling" OR "IO Mapping".DQ."Run Motor Cooling") AND NOT "CoolOverRunTimer".Q;
   "CoolOverRunTimer".TON(IN := #_w1 AND NOT "Request Run Motor Cooling", PT := "HMI Tags".CoolOverRunValue);
END_REGION
END_FUNCTION

FUNCTION "Analog Scaling" : Void   // FC7, LAD
{ S7_Optimized_Access := 'TRUE' }
// stored: SetENOAutomatically false
BEGIN

REGION Network 1: Line Pressure Scaling
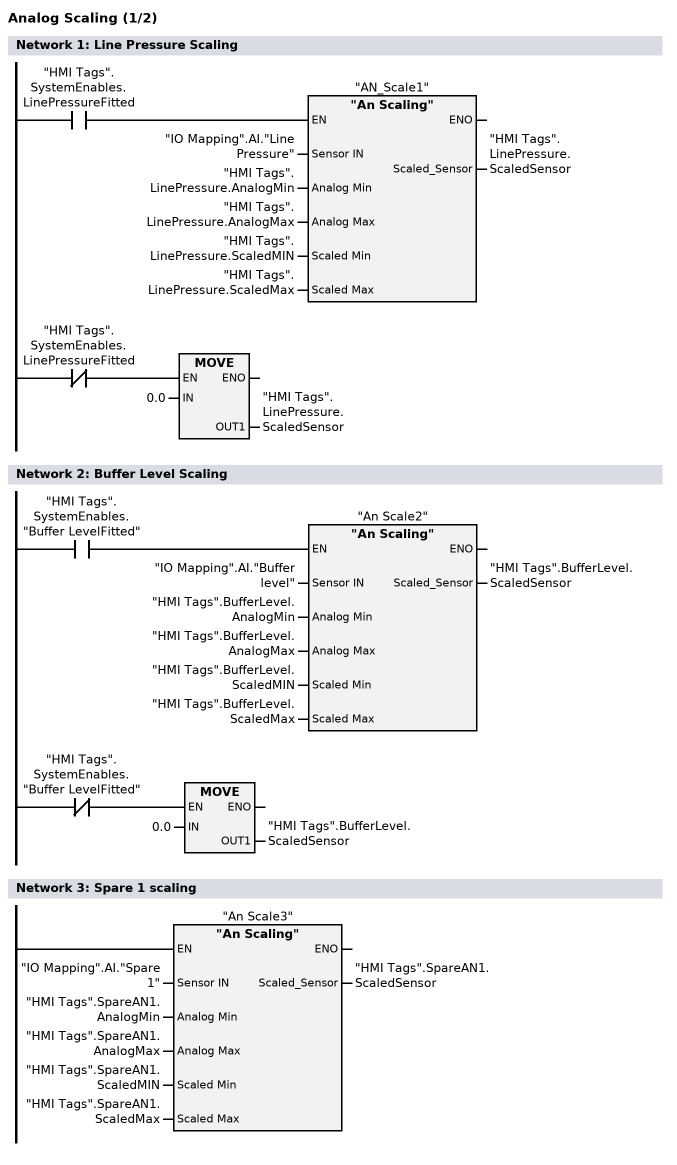
   RUNG wire#powerrail
      Contact( "HMI Tags".SystemEnables.LinePressureFitted )
      "AN_Scale1"("Sensor IN" := "IO Mapping".AI."Line Pressure", "Analog Min" := "HMI Tags".LinePressure.AnalogMin, "Analog Max" := "HMI Tags".LinePressure.AnalogMax, "Scaled Min" := "HMI Tags".LinePressure.ScaledMIN, "Scaled Max" := "HMI Tags".LinePressure.ScaledMax, Scaled_Sensor => "HMI Tags".LinePressure.ScaledSensor)
   END_RUNG
   RUNG wire#powerrail
      I_Contact( "HMI Tags".SystemEnables.LinePressureFitted )
      Move(in := 0.0, out1 => "HMI Tags".LinePressure.ScaledSensor)
   END_RUNG
   // the same network as SCL:
   IF "HMI Tags".SystemEnables.LinePressureFitted THEN
       "AN_Scale1"("Sensor IN" := "IO Mapping".AI."Line Pressure",   // "An Scaling"
                   "Analog Min" := "HMI Tags".LinePressure.AnalogMin,
                   "Analog Max" := "HMI Tags".LinePressure.AnalogMax,
                   "Scaled Min" := "HMI Tags".LinePressure.ScaledMIN,
                   "Scaled Max" := "HMI Tags".LinePressure.ScaledMax,
                   Scaled_Sensor => "HMI Tags".LinePressure.ScaledSensor);
   END_IF;
   IF NOT "HMI Tags".SystemEnables.LinePressureFitted THEN
       "HMI Tags".LinePressure.ScaledSensor := 0.0;
   END_IF;
END_REGION

REGION Network 2: Buffer Level Scaling
   RUNG wire#powerrail
      Contact( "HMI Tags".SystemEnables."Buffer LevelFitted" )
      "An Scale2"("Sensor IN" := "IO Mapping".AI."Buffer level", "Analog Min" := "HMI Tags".BufferLevel.AnalogMin, "Analog Max" := "HMI Tags".BufferLevel.AnalogMax, "Scaled Min" := "HMI Tags".BufferLevel.ScaledMIN, "Scaled Max" := "HMI Tags".BufferLevel.ScaledMax, Scaled_Sensor => "HMI Tags".BufferLevel.ScaledSensor)
   END_RUNG
   RUNG wire#powerrail
      I_Contact( "HMI Tags".SystemEnables."Buffer LevelFitted" )
      Move(in := 0.0, out1 => "HMI Tags".BufferLevel.ScaledSensor)
   END_RUNG
   // the same network as SCL:
   IF "HMI Tags".SystemEnables."Buffer LevelFitted" THEN
       "An Scale2"("Sensor IN" := "IO Mapping".AI."Buffer level",   // "An Scaling"
                   "Analog Min" := "HMI Tags".BufferLevel.AnalogMin,
                   "Analog Max" := "HMI Tags".BufferLevel.AnalogMax,
                   "Scaled Min" := "HMI Tags".BufferLevel.ScaledMIN,
                   "Scaled Max" := "HMI Tags".BufferLevel.ScaledMax,
                   Scaled_Sensor => "HMI Tags".BufferLevel.ScaledSensor);
   END_IF;
   IF NOT "HMI Tags".SystemEnables."Buffer LevelFitted" THEN
       "HMI Tags".BufferLevel.ScaledSensor := 0.0;
   END_IF;
END_REGION

REGION Network 3: Spare 1 scaling
   RUNG wire#powerrail
      "An Scale3"("Sensor IN" := "IO Mapping".AI."Spare 1", "Analog Min" := "HMI Tags".SpareAN1.AnalogMin, "Analog Max" := "HMI Tags".SpareAN1.AnalogMax, "Scaled Min" := "HMI Tags".SpareAN1.ScaledMIN, "Scaled Max" := "HMI Tags".SpareAN1.ScaledMax, Scaled_Sensor => "HMI Tags".SpareAN1.ScaledSensor)
   END_RUNG
   // the same network as SCL:
   "An Scale3"("Sensor IN" := "IO Mapping".AI."Spare 1",   // "An Scaling"
               "Analog Min" := "HMI Tags".SpareAN1.AnalogMin,
               "Analog Max" := "HMI Tags".SpareAN1.AnalogMax,
               "Scaled Min" := "HMI Tags".SpareAN1.ScaledMIN,
               "Scaled Max" := "HMI Tags".SpareAN1.ScaledMax,
               Scaled_Sensor => "HMI Tags".SpareAN1.ScaledSensor);
END_REGION

REGION Network 4: Spare 2 Scaling
